
// ===== library types =====

// folder: Library/Modbus/Core/Query

TYPE "mb_set_udt"
   STRUCT
      signed : Bool;   // Set true if it's a signed number.
      double : Bool;   // Get two trailing words (4 bytes) from buffer. False, get one word (2 bytes).
      factor : Real := 1.0;   // Factor the value from the buffer is multiplied with.
   END_STRUCT;
END_TYPE

// folder: Library/Modbus/Core/Sb

TYPE "mb_station_block_udt"
   STRUCT
      conf : Struct   // Configuration
         unit : USInt;   // mb_addr
         skip_code : Bool;   // Skip all code in header and footer fc's.
         disable : Bool;   // Skip all queries
         read_only : Bool;   // Skip all write queries. (fc 5,6,15,16)
         max_comm_error : USInt := 2;   // Repeating erros before communication_error flag is set
         exec_quantity : USInt := 1;   // Number of queries to be exec. at each loop.
      END_STRUCT;
      out : Struct   // Outputs
         Error : Bool;   // All errors, including communication errors
         Communication_error : Bool;   // only communication errors
         Finnish : Bool;   // qid is handed over to next device.
      END_STRUCT;
      log : Struct   // Logging for development and debugging.
         Connected_time : DTL;   // The time the device was connected to the bus
         Disconnected_time : DTL;   // The time, if a device was disconnected to the bus
         Done_cnt : UDInt;   // Successfully queries counter for this device
         Error_comm_cnt : UDInt;   // Communication erros cnt.
         Error_exception_cnt : UDInt;   // Failed queries counter for this device
         Error_status : Word;   // Status code from mb_master or mb_client
         Error_data_addr : UDInt;   // d_addr for last failed querie; handy for troubleshooting
      END_STRUCT;
      z : Struct   // Internal states.
         header_qid : UInt;   // qid value at device header
         comm_err_cnt : USInt;   // Repeating communication errors
         exec_cnt : USInt;   // Numb. of exec. q. this loop
         offset_qid : UInt := 1;   // Device query id.
         err_hold : Bool;   // Help var for .out.error
      END_STRUCT;
   END_STRUCT;
END_TYPE

// folder: Library/Modbus/Core/Tcp

TYPE "mb_tcp_connection_udt"
   STRUCT
      ip : Array[1..4] of USInt;   // IP address
      tcp_port : UInt := 502;
      timeout : Time;
      Error : Bool;
      Error_network : Bool;   // Error with network connection
      Error_unit : USInt;   // Device with error
      z : Struct   // Internal variables
         qid_bellow : Bool;
         disconnect : Bool;   // This tcp-connection has disconnected the connection.
         init_at_header : Bool;   // True if run-state is INIT_QUERY at the header.
      END_STRUCT;
   END_STRUCT;
END_TYPE

// folder: Library/Modbus/Station blocks/sb Untested/M/Mettler

TYPE "mettlerToledoInd560Udt"
   STRUCT
      readMsgSlot : Array[1..4] of Struct
         cmdRespons : Struct
            FP_1 : Bool;
            FP_2 : Bool;
            FP_3 : Bool;
            FP_4 : Bool;
            FP_5 : Bool;
            data_integrity : Bool;
            cmdAck1 : Bool;
            cmdAck2 : Bool;
         END_STRUCT;
         reserved : Byte;   // volt
         data : Real;
         scale_status : Struct
            x08_Enter_Key : Bool;
            x09_Input_1 : Bool;
            x10_Input_2 : Bool;
            x11_Input_3 : Bool;
            x12_Motion : Bool;
            x13_Net_Mode : Bool;
            x14_Data_Integrity_2 : Bool;
            x15_Data_OK : Bool;
            x00_Target_1 : Bool;
            x01_Comparator_1 : Bool;
            x02_Targe_2 : Bool;
            x03_Comparator_2 : Bool;
            x04_Target_3 : Bool;
            x05_Alway_true : Bool;
            x06_TE_bit_1 : Bool;
            x07_TE_bit_2 : Bool;
         END_STRUCT;
      END_STRUCT;
      writeMsgSlot : Array[1..4] of Struct
         cmd : UInt;
         data : Real;
      END_STRUCT;
      run : Struct   // Data calculated from readMsgSlot
         PF : Array[1..4] of USInt;   // Floating point input indication
         cmdAck : Array[1..4] of USInt;
      END_STRUCT;
      occupiedMsgSlots : Array[1..4] of Bool;
      queryDone : Struct
         read : Bool;
         write : Bool;
      END_STRUCT;
   END_STRUCT;
END_TYPE

// folder: Library/Modbus/Station blocks/udt interfaces

TYPE "energy_udt"
   STRUCT
      current : Struct
         L : Array[1..3] of Real;   // A - Live
         N : Real;   // A - Neutral
         avg : Real;   // A - Average
      END_STRUCT;
      voltage : Struct
         L_L : Array[1..3] of Real;   // V
         L_L_avg : Real;   // V - Average
         L_N : Array[1..3] of Real;   // V
         L_N_avg : Real;   // V - Average
      END_STRUCT;
      power : Struct
         active : Struct
            L : Array[1..3] of Real;   // kW
            total : Real;   // kW
         END_STRUCT;
         reactive : Struct
            L : Array[1..3] of Real;   // kVAR
            total : Real;   // kVAR
         END_STRUCT;
         apparent : Struct
            L : Array[1..3] of Real;   // kVA
            total : Real;   // kVA
         END_STRUCT;
      END_STRUCT;
      energy : Struct   // (Accumulated)
         active_out : Real;   // kWh - delivered
         active_in : Real;   // kWh - received
         reactive_out : Real;   // kVARh
         reactive_in : Real;   // kVARh
         apparent_out : Real;   // kVAh
         apparent_in : Real;   // kVAh
      END_STRUCT;
      reverse_phase_order : Bool;
   END_STRUCT;
   // // voltage.L_L[1] : V
END_TYPE

TYPE "variable_frequency_drive_udt"
   STRUCT
      in : Struct   // Input
         ref : Real;   // %
         start : Bool;
         cost : Bool;
         dc_break : Bool;
         quick_stop : Bool;
         reset : Bool;
      END_STRUCT;
      out : Struct   // Output
         ready : Bool;   // Whating only for start signal from plc
         auto : Bool;   // Auto on keypad of device.
         in_operation : Bool;   // Device is operation.
         running : Bool;   // Motor is spinning
         error : Bool;
         power : Real;   // [kW]
         current : Real;   // [A]
         voltage : Real;   // [V]
         frequency : Real;   // [Hz]
         rpm : Real;   // Revolutions per minute
         output_percent : Real;
         torque_percent : Real;
         heatsing_temperature : Real;   // degrees celsius
      END_STRUCT;
   END_STRUCT;
END_TYPE

TYPE "flow_udt"
   STRUCT
      volume_flow : Real;   // kg/s
      mass_flow : Real;   // m3/s
      velocity : Real;   // m/s
      density : Real;   // kg/m3
      temperature : Real;   // °C
   END_STRUCT;
END_TYPE

// folder: Library/Modbus/.Start examples

FUNCTION "mb_Readme" : Void   // FC13, SCL
{ S7_Optimized_Access := 'TRUE' }
VERSION : 0.1
BEGIN
   (* Instructions:

   - Add one of the exmple FB's to your PLC.
   - Call that FB from a cyclic OB.
   - Terminate connection to type on the example FB. (Right click the FB)
   - Set hardware_id, buad-rate, ip, tcp-port, etc, to the correct value.
   - Look inside the library and check if there is a ready station block (SB),
     for your program. If there isn't then a new has to be made. 
   - Station blocks can be single-DB's or multi-instances in a FB.
   - Remove the exmple code and example SB's.

     IMPORTANT: As stated above, the start examples fb, need to be terminated 
     from the library type. If the type is edited and later there is a library 
     update, then all the changes will get lost.

   - Instructions need to be set to the latest version: (Usually already okay)
      * Instructions -> Communication -> Others -> Modbus TCP
      * Instructions -> Communication -> Communication processor -> Modbus
      * Instructions -> Communication -> Communication processor -> Modbus (RTU)  
      * Instructions -> Basic instructions -> Word logic operations -> SEL.
     Change version in the right column.

   *)
END_FUNCTION

// folder: Library/Modbus/.Start examples/Rtu/1200

FUNCTION_BLOCK "modbus_rtu_1200"   // FB104, SCL
{ S7_Optimized_Access := 'TRUE' }
VERSION : 0.1
   VAR
      mb_query : "mb_query";
      mb_rtu1200_ctrl : "mb_rtu1200_ctrl";
      abb_aquaMaster_device1 : "abb_aquaMaster_3";
      abb_aquaMaster_device2 : "abb_aquaMaster_3";
      abb_aquaMaster_device3 : "abb_aquaMaster_3";
      Auma_valve : "Auma_valve";
      Phoenix_Contact_UPS : "Phoenix_Contact_UPS";
      resault_data : Word;
   END_VAR
BEGIN
   // hardware_id: Can be found inside "Device configuration".
   // baud:        Bits per sec. (Parity is even by default)
   // mb_query:    The FB that connects everything together.
   #mb_rtu1200_ctrl(hardware_id := 0, // REPLACE WITH CORRECT ID.
                    baud := 19200,
                    mb_query := #mb_query);

   // - Timeout is calculated automatically.
   // - Each blocks bellow represent one device on the bus.

   // Three Abb aqua-master's.
   #abb_aquaMaster_device1(mb_addr := 1, mb_query := #mb_query);
   #abb_aquaMaster_device2(mb_addr := 2, mb_query := #mb_query);
   #abb_aquaMaster_device3(mb_addr := 3, mb_query := #mb_query);

   // A valve 
   #Auma_valve(mb_addr := 4, mb_query := #mb_query);

   // A UPS.
   #Phoenix_Contact_UPS(mb_addr := 5, mb_query := #mb_query);

   // A station block can be used both for both modbus rtu and tcp. This
   // is particular useful if a tcp-rtu-gateway is used. The same program
   // could be used, just swap mb_master_1200_ctrl, with mb_client_ctrl.

   // Read holding register 456 from device with modbus address 123.
   // This is an example showing that a query does not necessarily need
   // to be part of a station block (SB) as obove, however making
   // reusable SB's is good practice.
   #mb_query(mb_addr := 123,
             mode := #mb_query.c.read.holding_reg,
             data_addr := 456,
             data_ptr := #resault_data);


   // Debugging tip, (no code)
   "mb_Debugging"();
END_FUNCTION_BLOCK

FUNCTION_BLOCK "modbus_rtu_1200_ladder"   // FB114, LAD
TITLE = Example modbus rtu
{ S7_Optimized_Access := 'TRUE' }
VERSION : 0.1
   VAR
      mb_master_ctrl : "mb_rtu1200_ctrl";
      mb_query : "mb_query";
      aquaMaster_device1 : "abb_aquaMaster_3";
      aquaMaster_device2 : "abb_aquaMaster_3";
      Auma_valve : "Auma_valve";
      Phoenix_Contact_UPS : "Phoenix_Contact_UPS";
   END_VAR
   VAR_TEMP   // added for the SCL form of the ladder/FBD networks
      _w1 : Bool;
   END_VAR
BEGIN

REGION Network 1: Modbus master
   // Replace 'hardware_id' with correct id.
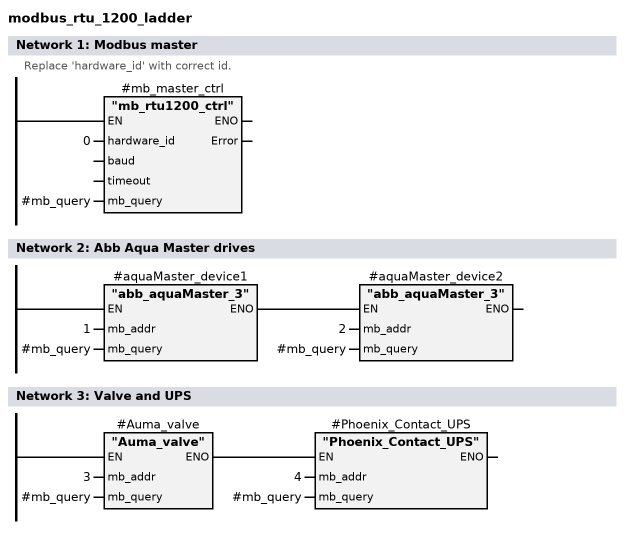
   RUNG wire#powerrail
      #mb_master_ctrl(hardware_id := 0, baud :=, mb_query := #mb_query, Error =>, timeout :=)
   END_RUNG
   // the same network as SCL:
   #mb_master_ctrl(hardware_id := 0, mb_query := #mb_query);   // "mb_rtu1200_ctrl"
END_REGION

REGION Network 2: Abb Aqua Master drives
   RUNG wire#powerrail
      #aquaMaster_device1(mb_addr := 1, mb_query := #mb_query)
      #aquaMaster_device2(mb_addr := 2, mb_query := #mb_query)
   END_RUNG
   // the same network as SCL:
   #aquaMaster_device1(mb_addr := 1, mb_query := #mb_query, ENO => #_w1);   // "abb_aquaMaster_3"
   IF #_w1 THEN
       #aquaMaster_device2(mb_addr := 2, mb_query := #mb_query);   // "abb_aquaMaster_3"
   END_IF;
END_REGION

REGION Network 3: Valve and UPS
   RUNG wire#powerrail
      #Auma_valve(mb_addr := 3, mb_query := #mb_query)
      #Phoenix_Contact_UPS(mb_addr := 4, mb_query := #mb_query)
   END_RUNG
   // the same network as SCL:
   #Auma_valve(mb_addr := 3, mb_query := #mb_query, ENO => #_w1);   // "Auma_valve"
   IF #_w1 THEN
       #Phoenix_Contact_UPS(mb_addr := 4, mb_query := #mb_query);   // "Phoenix_Contact_UPS"
   END_IF;
END_REGION
END_FUNCTION_BLOCK

FUNCTION_BLOCK "modbus_rtu_1200_empty"   // FB119, SCL
{ S7_Optimized_Access := 'TRUE' }
VERSION : 0.1
   VAR
      mb_query : "mb_query";
      mb_master_1200_ctrl : "mb_rtu1200_ctrl";
      _ : Bool;
   END_VAR
BEGIN
   // hardware_id: Can be found inside "Device configuration".
   // baud:        Bits per sec. (Parity is even by default)
   // mb_query:    The FB that connects everything together.
   #mb_master_1200_ctrl(hardware_id := 0, // REPLACE WITH CORRECT ID. ("Local~CB_1241_(RS485)")
                        baud := 19200,
                        mb_query := #mb_query);

   // Timeout is calculated automatically.

   // ... Insert station blocks here ...



   // Debugging tip, (no code)
   "mb_Debugging"();
END_FUNCTION_BLOCK

// folder: Library/Modbus/.Start examples/Rtu/1500

FUNCTION_BLOCK "modbus_rtu_1500_empty"   // FB5, SCL
{ S7_Optimized_Access := 'TRUE' }
VERSION : 0.1
   VAR
      mb_query : "mb_query";
      mb_rtu1500_ctrl : "mb_rtu1500_ctrl";
      _ : Bool;
   END_VAR
BEGIN
   // hardware_id:     May be found inside the hardware configuration.
   // operating_mode:  0: RS232, 2: RS422, 4: RS485.
   // baud:            Bits per sec. (Parity is even by default)
   // mb_query:        The FB that connects everything together.
   #mb_rtu1500_ctrl(hardware_id := 0, // REPLACE WITH CORRECT ID.
                    operating_mode := 4, // RS-485
                    baud := 19200, // bps
                    mb_query := #mb_query);

   // Timeout is calculated automatically.


   // ... Insert station blocks here ...



   // Debugging tip, (no code)
   "mb_Debugging"();
END_FUNCTION_BLOCK

FUNCTION_BLOCK "modbus_rtu_1500_ladder"   // FB97, LAD
TITLE = Example modbus rtu for S7-1500
{ S7_Optimized_Access := 'TRUE' }
VERSION : 0.1
   VAR
      mb_rtu1500_ctrl : "mb_rtu1500_ctrl";
      mb_query : "mb_query";
      aquaMaster_device1 : "abb_aquaMaster_3";
      aquaMaster_device2 : "abb_aquaMaster_3";
      Auma_valve : "Auma_valve";
      Phoenix_Contact_UPS : "Phoenix_Contact_UPS";
   END_VAR
   VAR_TEMP   // added for the SCL form of the ladder/FBD networks
      _w1 : Bool;
   END_VAR
BEGIN

REGION Network 1: Modbus master
   // hardware_id:            Can be found inside "Device configuration". 
   // operating_mode:    0: RS232, 2: RS422, 4: RS485.
   // baud:                         Bits per sec. (Parity is even by default)
   // mb_query:                The FB that connects everything together.
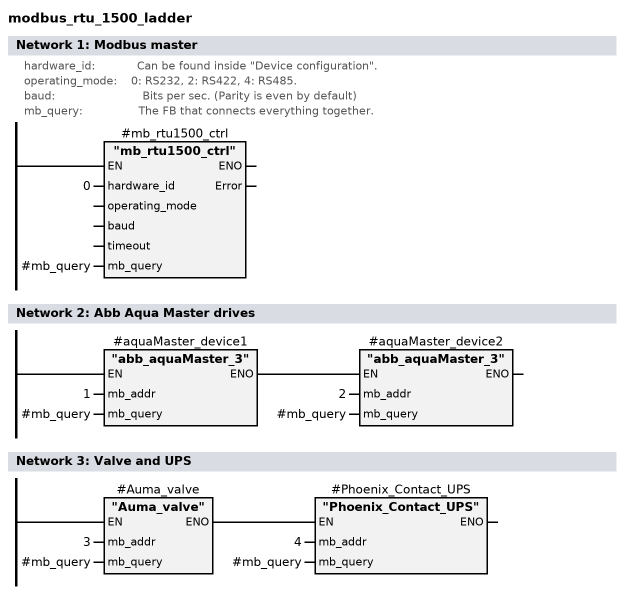
   RUNG wire#powerrail
      #mb_rtu1500_ctrl(hardware_id := 0, operating_mode :=, baud :=, timeout :=, mb_query := #mb_query, Error =>)
   END_RUNG
   // the same network as SCL:
   #mb_rtu1500_ctrl(hardware_id := 0, mb_query := #mb_query);   // "mb_rtu1500_ctrl"
END_REGION

REGION Network 2: Abb Aqua Master drives
   RUNG wire#powerrail
      #aquaMaster_device1(mb_addr := 1, mb_query := #mb_query)
      #aquaMaster_device2(mb_addr := 2, mb_query := #mb_query)
   END_RUNG
   // the same network as SCL:
   #aquaMaster_device1(mb_addr := 1, mb_query := #mb_query, ENO => #_w1);   // "abb_aquaMaster_3"
   IF #_w1 THEN
       #aquaMaster_device2(mb_addr := 2, mb_query := #mb_query);   // "abb_aquaMaster_3"
   END_IF;
END_REGION

REGION Network 3: Valve and UPS
   RUNG wire#powerrail
      #Auma_valve(mb_addr := 3, mb_query := #mb_query)
      #Phoenix_Contact_UPS(mb_addr := 4, mb_query := #mb_query)
   END_RUNG
   // the same network as SCL:
   #Auma_valve(mb_addr := 3, mb_query := #mb_query, ENO => #_w1);   // "Auma_valve"
   IF #_w1 THEN
       #Phoenix_Contact_UPS(mb_addr := 4, mb_query := #mb_query);   // "Phoenix_Contact_UPS"
   END_IF;
END_REGION
END_FUNCTION_BLOCK

FUNCTION_BLOCK "modbus_rtu_1500"   // FB108, SCL
{ S7_Optimized_Access := 'TRUE' }
VERSION : 0.1
   VAR
      mb_query : "mb_query";
      mb_rtu1500_ctrl : "mb_rtu1500_ctrl";
      abb_aquaMaster_device1 : "abb_aquaMaster_3";
      abb_aquaMaster_device2 : "abb_aquaMaster_3";
      abb_aquaMaster_device3 : "abb_aquaMaster_3";
   END_VAR
BEGIN
   // hardware_id:     May be found inside the hardware configuration.
   // operating_mode:  0: RS232, 2: RS422, 4: RS485.
   // baud:            Bits per sec. (Parity is even by default)
   // mb_query:        The FB that connects everything together.
   #mb_rtu1500_ctrl(hardware_id := 0, // REPLACE WITH CORRECT ID.
                    operating_mode := 4, // RS-485
                    baud := 19200, // bps
                    mb_query := #mb_query);

   // Timeout is calculated automatically

   // Each blocks bellow represent one device on the bus. 
   #abb_aquaMaster_device1(mb_addr := 1, mb_query := #mb_query);
   #abb_aquaMaster_device2(mb_addr := 2, mb_query := #mb_query);
   #abb_aquaMaster_device3(mb_addr := 3, mb_query := #mb_query);


   // Debugging tip, (no code)
   "mb_Debugging"();
END_FUNCTION_BLOCK

// folder: Library/Modbus/.Start examples/Tcp

FUNCTION_BLOCK "modbus_tcp_empty"   // FB79, SCL
{ S7_Optimized_Access := 'TRUE' }
VERSION : 0.1
   VAR
      mb_query : "mb_query";
      mb_client_ctrl : "mb_tcp_ctrl";
      ip : Array[1..4] of USInt;
      mb_delay_between_queries : "mb_delay_between_queries";
   END_VAR
BEGIN
   // IP-address of the modbus server
   #ip[1] := 192;
   #ip[2] := 168;
   #ip[3] := 1;
   #ip[4] := 2;

   // interface:  Profinet interface.
   //             (Find const. inside "Device configuration")
   // conn_id:    A unique id for each tcp connectin in the plc.
   // ip_addr:    The ip-address of the server. (Array of 4 bytes)
   // tcp_port:   Default port is 502. (UDP isn't available)
   // timeout:    Depends on the network conncetion.
   // mb_query:   The query FB.
   #mb_client_ctrl(interface := 0, // REPLACE WITH CORRECT ID OR CONST,
                                   // Eg. "Local~PROFINET_interface_1",
                   conn_id := 123,
                   ip_addr := #ip,
                   tcp_port := 502,
                   timeout := T#2s,
                   mb_query := #mb_query);

   // Delay the query execution, this prevent the plc from
   // jamming the network. Adjust the time to the application.
   #mb_delay_between_queries(delay := T#500ms,
                             mb_query := #mb_query);




   // ... Insert station blocks here ...




   // Debugging tip, (no code)
   "mb_Debugging"();
END_FUNCTION_BLOCK

FUNCTION_BLOCK "modbus_tcp_ladder"   // FB98, LAD
TITLE = Example modbus tcp
{ S7_Optimized_Access := 'TRUE' }
VERSION : 0.1
   VAR
      mb_client_ctrl : "mb_tcp_ctrl";
      mb_query : "mb_query";
      mb_delay_between_queries : "mb_delay_between_queries";
      ip : Array[1..4] of USInt;
      siemens_PAC3200 : "Siemens_PAC3200";
   END_VAR
   VAR_TEMP   // added for the SCL form of the ladder/FBD networks
      _w1 : Bool;
   END_VAR
BEGIN

REGION Network 1 (SCL): IP-address
   #ip[1] := 192;
   #ip[2] := 168;
   #ip[3] := 1;
   #ip[4] := 123;
END_REGION

REGION Network 2: Modbus client ctrl
   // - Insert interface constant, eg "Local~PROFINET_interface_1". 
   // - conn_id need to be unique for all tcp connection in the plc.
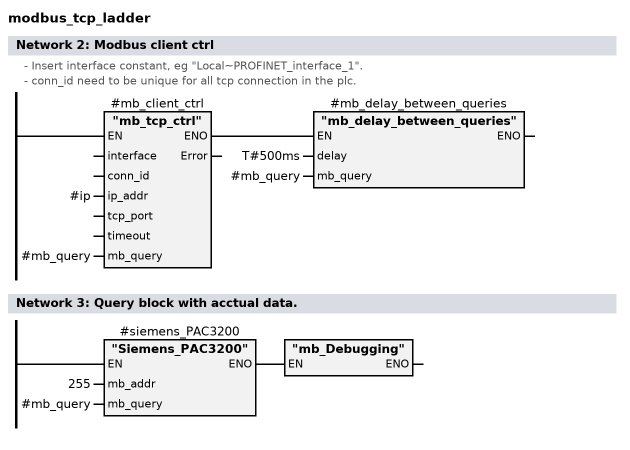
   RUNG wire#powerrail
      #mb_client_ctrl(interface :=, conn_id :=, ip_addr := #ip, tcp_port :=, timeout :=, mb_query := #mb_query, Error =>)
      #mb_delay_between_queries(delay := T#500ms, mb_query := #mb_query)
   END_RUNG
   // the same network as SCL:
   #mb_client_ctrl(ip_addr := #ip, mb_query := #mb_query, ENO => #_w1);   // "mb_tcp_ctrl"
   IF #_w1 THEN
       #mb_delay_between_queries(delay := T#500ms, mb_query := #mb_query);   // "mb_delay_between_queries"
   END_IF;
END_REGION

REGION Network 3: Query block with acctual data.
   RUNG wire#powerrail
      #siemens_PAC3200(mb_addr := 255, mb_query := #mb_query)
      "mb_Debugging"()
   END_RUNG
   // the same network as SCL:
   #siemens_PAC3200(mb_addr := 255, mb_query := #mb_query, ENO => #_w1);   // "Siemens_PAC3200"
   IF #_w1 THEN "mb_Debugging"(); END_IF;
END_REGION
END_FUNCTION_BLOCK

FUNCTION_BLOCK "modbus_tcp"   // FB110, SCL
{ S7_Optimized_Access := 'TRUE' }
VERSION : 0.1
   VAR
      mb_query : "mb_query";
      mb_tcp_ctrl : "mb_tcp_ctrl";
      siemens_PAC3200 : "Siemens_PAC3200";
      ip : Array[1..4] of USInt;
      mb_delay_between_queries : "mb_delay_between_queries";
   END_VAR
BEGIN
   // IP-address of the modbus server
   #ip[1] := 192;
   #ip[2] := 168;
   #ip[3] := 1;
   #ip[4] := 2;

   // interface:  Profinet interface.
   //             (Find const. inside "Device configuration")
   // conn_id:    A unique id for each tcp connectin in the plc.
   // ip_addr:    The ip-address of the server. (Array of 4 bytes)
   // tcp_port:   Default port is 502. (UDP isn't available)
   // timeout:    Depends on the network conncetion.
   // mb_query:   The query FB.
   #mb_tcp_ctrl(interface := 0, // REPLACE WITH CORRECT ID OR CONST,
                // Eg. "Local~PROFINET_interface_1",
                conn_id := 123,
                ip_addr := #ip,
                tcp_port := 502,
                timeout := T#2s,
                mb_query := #mb_query);

   // Delay the query execution, this prevent the plc from
   // jamming the network. Adjust the time to the application.
   #mb_delay_between_queries(delay := T#500ms, mb_query := #mb_query);

   #siemens_PAC3200(mb_query := #mb_query);


   // Debugging tip, (no code)
   "mb_Debugging"();
END_FUNCTION_BLOCK

// folder: Library/Modbus/.Start examples/Tcp/multi_client

FUNCTION_BLOCK "multi_client"   // FB111, SCL
{ S7_Optimized_Access := 'TRUE' }
VERSION : 0.1
   VAR
      ctrl : "mb_tcp_ctrl";
      query : "mb_query";
      delay_between_queries : "mb_delay_between_queries";
      c1 : "mb_tcp_connection_udt";
      c2 : "mb_tcp_connection_udt";
      c3 : "mb_tcp_connection_udt";
      c4 : "mb_tcp_connection_udt";
      c5 : "mb_tcp_connection_udt";
      power_meter_1 : "Siemens_PAC3200";
      power_meter_2 : "Siemens_PAC3200";
      flow_meter_1 : "Siemens_MAG_6000";
      flow_meter_2 : "Siemens_MAG_6000";
      Level_1 : "Mjk_expert";
      Level_2 : "Mjk_expert";
      Level_3 : "Mjk_expert";
   END_VAR
BEGIN
   // This feature is foremost intended for S7-1200 where the number of tcp
   // connections is limited. Another use case it's to get data from hundreds or 
   // even tunsens of devices, and it's then also applicable for S7-1500 plc's.
   // One mb_client use much memory, so you would save memory by using this
   // approach, compare using a client for each connection.
   //
   // One mb_client is connecting and disconnecting to different ip-addresses,
   // and therefore only occupy one connection. The downside with this solution
   // is the delays for data to come in. The library is smart, and it wouldn't
   // waste time on polling devices that has got timeout before.

   // Important: Don't assign anything to #ctrl.ip_addr and #ctrl.tcp_port, when
   //            the library is used in this mode.

   // interface:  Profinet interface. (Find const. inside "Device configuration")
   // conn_id:    A unique id for each tcp connectin in the plc.
   // timeout:    Establish a tcp-connection may take quite long, several
   //             seconds for some devices, so make sure to not set it to short.
   // mb_query:   The query FB.
   #ctrl(interface := 64, conn_id := 123, timeout := T#2s, mb_query := #query);

   // Delay the query execution, this prevent the plc from
   // jamming the network. Adjust the time to the application.
   #delay_between_queries(delay := T#20ms, mb_query := #query);

   REGION TCP-connection 1
       #c1.ip[1] := 192;
       #c1.ip[2] := 168;
       #c1.ip[3] := 0;
       #c1.ip[4] := 2;
       "mb_tcp_connection_header"(conn := #c1, ctrl := #ctrl, q := #query);

       // Note: For some tcp-devices mb_addr need to be set to 255.
       #power_meter_1(mb_query := #query);

       "mb_tcp_connection_foother"(conn := #c1, ctrl := #ctrl, q := #query);
   END_REGION

   REGION TCP-connection 2
       #c2.ip[1] := 192;
       #c2.ip[2] := 168;
       #c2.ip[3] := 0;
       #c2.ip[4] := 3;
       "mb_tcp_connection_header"(conn := #c2, ctrl := #ctrl, q := #query);

       #power_meter_2(mb_query := #query);

       "mb_tcp_connection_foother"(conn := #c2, ctrl := #ctrl, q := #query);
   END_REGION

   REGION TCP-connection 3
       #c3.ip[1] := 192;
       #c3.ip[2] := 168;
       #c3.ip[3] := 0;
       #c3.ip[4] := 4;
       "mb_tcp_connection_header"(conn := #c3, ctrl := #ctrl, q := #query);

       #flow_meter_1(mb_query := #query);

       "mb_tcp_connection_foother"(conn := #c3, ctrl := #ctrl, q := #query);
   END_REGION

   REGION TCP-connection 4
       #c4.ip[1] := 192;
       #c4.ip[2] := 168;
       #c4.ip[3] := 0;
       #c4.ip[4] := 5;
       "mb_tcp_connection_header"(conn := #c4, ctrl := #ctrl, q := #query);

       #flow_meter_2(mb_query := #query);

       "mb_tcp_connection_foother"(conn := #c4, ctrl := #ctrl, q := #query);
   END_REGION

   REGION TCP-connection 5 (gateway)
       #c5.ip[1] := 192;
       #c5.ip[2] := 168;
       #c5.ip[3] := 0;
       #c5.ip[4] := 6;
       "mb_tcp_connection_header"(conn := #c5, ctrl := #ctrl, q := #query);

       // For a gateway, any number of station blocks may be placed between
       // header above and the foother bellow.
       #Level_1(mb_addr := 1, mb_query := #query);
       #Level_2(mb_addr := 2, mb_query := #query);
       #Level_3(mb_addr := 3, mb_query := #query);

       "mb_tcp_connection_foother"(conn := #c5, ctrl := #ctrl, q := #query);
   END_REGION

   "mb_Debugging"(); // Just text.
END_FUNCTION_BLOCK

FUNCTION_BLOCK "multi_client_empty"   // FB118, SCL
{ S7_Optimized_Access := 'TRUE' }
VERSION : 0.1
   VAR
      ctrl : "mb_tcp_ctrl";
      query : "mb_query";
      delay_between_queries : "mb_delay_between_queries";
      c1 : "mb_tcp_connection_udt";
      c2 : "mb_tcp_connection_udt";
      c3 : "mb_tcp_connection_udt";
   END_VAR
BEGIN

   // interface:  Profinet interface. (Find const. inside "Device configuration")
   // conn_id:    A unique id for each tcp connectin in the plc.
   // timeout:    Establish a tcp-connection may take quite long, serveral
   //             secounds for some devices, so make sure to not set it to short.
   //             On the other hand it's also important to set it too long.
   //             On a local network you may try to start with 3 sec.
   // mb_query:   The query FB.                                     
   #ctrl(interface := 64, conn_id := 123, timeout := T#3s, mb_query := #query);

   // Delay the query execution, this prevent the plc from
   // jamming the network. Adjust the time to the application.
   #delay_between_queries(delay := T#50ms, mb_query := #query);

   REGION TCP-connection 1
       #c1.ip[1] := 192;
       #c1.ip[2] := 168;
       #c1.ip[3] := 0;
       #c1.ip[4] := 0;
       "mb_tcp_connection_header"(conn := #c1, ctrl := #ctrl, q := #query);

       // Insert sb here.

       "mb_tcp_connection_foother"(conn := #c1, ctrl := #ctrl, q := #query);
   END_REGION

   REGION TCP-connection 2
       #c2.ip[1] := 192;
       #c2.ip[2] := 168;
       #c2.ip[3] := 0;
       #c2.ip[4] := 0;
       "mb_tcp_connection_header"(conn := #c2, ctrl := #ctrl, q := #query);

       // Insert sb here.

       "mb_tcp_connection_foother"(conn := #c2, ctrl := #ctrl, q := #query);
   END_REGION

   REGION TCP-connection 3
       #c3.ip[1] := 192;
       #c3.ip[2] := 168;
       #c3.ip[3] := 0;
       #c3.ip[4] := 0;
       "mb_tcp_connection_header"(conn := #c3, ctrl := #ctrl, q := #query);

       // Insert sb here.

       "mb_tcp_connection_foother"(conn := #c3, ctrl := #ctrl, q := #query);
   END_REGION


   "mb_Debugging"(); // Only text
END_FUNCTION_BLOCK

FUNCTION_BLOCK "multi_client_array"   // FB121, SCL
{ S7_Optimized_Access := 'TRUE' }
VERSION : 0.1
   VAR
      ctrl : "mb_tcp_ctrl";
      query : "mb_query";
      delay_between_queries : "mb_delay_between_queries";
      c : Array[2..50] of "mb_tcp_connection_udt";
      power_meter : Array[2..50] of "Siemens_PAC3200";
      j : Int := 2;
   END_VAR
BEGIN
   // An example with many tcp devices.

   // interface:  Profinet interface. (Find const. inside "Device configuration")
   // conn_id:    A unique id for each tcp connectin in the plc.
   // timeout:    Establish a tcp-connection may take quite long, serveral
   //             secounds for some devices, so make sure to not set it to short. 
   // mb_query:   The query FB.                                     
   #ctrl(interface := 64, conn_id := 123, timeout := T#2s, mb_query := #query);

   // Delay the query execution, this prevent the plc from
   // jamming the network. Adjust the time to the application.
   #delay_between_queries(delay := T#20ms, mb_query := #query);

   #c[#j].ip[1] := 192;
   #c[#j].ip[2] := 168;
   #c[#j].ip[3] := 0;
   #c[#j].ip[4] := INT_TO_USINT(#j);
   "mb_tcp_connection_header"(conn := #c[#j], ctrl := #ctrl, q := #query);

   #power_meter[#j]power_meter(mb_query := #query);

   "mb_tcp_connection_foother"(conn := #c[#j], ctrl := #ctrl, q := #query);

   #j += BOOL_TO_INT(#power_meter[#j].sb.out.Finnish);
   IF #j > 50 THEN
       #j := 2;
   END_IF;

   "mb_Debugging"(); // Just text.
END_FUNCTION_BLOCK

// folder: Library/Modbus/Core/Ctrl

FUNCTION_BLOCK "mb_tcp_ctrl"   // FB9, SCL
{ S7_Optimized_Access := 'TRUE' }
VERSION : 1.0
   VAR_INPUT
      interface : Hw_Any := 64;   // Profinet interface id
      conn_id : Conn_Ouc := 123;   // Connection id. Should be unique between all tcp connections.
      ip_addr : Array[1..4] of USInt;   // IPv4 address.
      tcp_port : UInt := 502;
      timeout : Time := T#3s;
   END_VAR
   VAR_OUTPUT
      Error : Bool;   // error flag with tof timer
   END_VAR
   VAR_IN_OUT
      mb_query : "mb_query";   // udt mb
   END_VAR
   VAR
      conf : Struct   // Configuration that normal shouldn't need to be changed.
         disconnect : Bool := false;
         retries : USInt := 0;
         timeout_connect : Time;   // May be set longer, then the main timeout. T#0s => Use normal timeout.
         disconnect_on_80A3 : Bool := true;
         fast_err : Bool := true;
      END_STRUCT;
      client : MB_CLIENT;
      tcon_ip_v4 : TCON_IP_v4;
      tdiscon : TDISCON;
      ton_timeout : TON_TIME;
      end : "mb_internal_e";
      override_timeout : Time;
      connected_memory : Bool;
      connected : Bool;
   END_VAR
   VAR_TEMP
      comm_err : Bool;
      c : SInt;
      t : Time;   // Timeout
   END_VAR
   VAR CONSTANT
      INIT_QUERY : USInt := 2;
      EXEC_QUERY : USInt := 3;
   END_VAR
BEGIN
   // Rexhip - Extended modbus library.
   //
   // Modbus tcp for S7-1200 and S7-1500.

   REGION Init
       // InterfaceId can be found inside "Device configuration".
       #tcon_ip_v4.InterfaceId := #interface;
       #tcon_ip_v4.ID := #conn_id; // Connection id
       FOR #c := 1 TO 4 DO // usint easier to read ip in plc-monitoring.
           #tcon_ip_v4.RemoteAddress.ADDR[#c] := USINT_TO_BYTE(#ip_addr[#c]); 
       END_FOR;
       #tcon_ip_v4.RemotePort := #tcp_port;
       #tcon_ip_v4.ConnectionType := 11; // tcp
       #tcon_ip_v4.ActiveEstablished := true; // Client

       IF #conf.disconnect THEN // Reset memory
           #connected_memory := false;  
       END_IF;

       IF #mb_query.z.run.state = #INIT_QUERY THEN
           RESET_TIMER(#ton_timeout);

           // Conversion of function codes.     
           "mb_internal_a"(Mode => #client.MB_MODE,
                           Data_addr => #client.MB_DATA_ADDR,
                           mb_query := #mb_query);
           #client.MB_Unit_ID := UINT_TO_BYTE(#mb_query.z.q.mb_addr);
           #client.Retries := #conf.retries;
           // Reset all stat-flags.
           #mb_query.stat.error := #mb_query.stat.error_comm :=
           (* *)#mb_query.stat.done := false;

           #mb_query.z.run.state := #EXEC_QUERY; // Next state.
       END_IF;
   END_REGION

   REGION Timeout
       IF #override_timeout <> T#0s THEN
           // If a value has been set for multi connection.
           #t := #override_timeout;
           #override_timeout := T#0s;
       ELSE
           // Use #timeout if #timeout_connect is set to zero. 
           // and connection has not been established before.
           #t := SEL(G := #conf.timeout_connect <> T#0s
                     AND NOT #connected_memory,
                     IN0 := #timeout,
                     IN1 := #conf.timeout_connect);
       END_IF;
       #t := LIMIT(MN := t#100ms, IN := #t, MX := t#10S);
       // If mb_client does not establish a connection it will not throw
       // timeout error. Timeout is handled manually for that case. 
       PRESET_TIMER(PT := #t,
                    TIMER := #ton_timeout);
       #client.Rcv_Timeout := UDINT_TO_REAL(T_CONV(#t)) * 0.001;
       #ton_timeout(IN := #mb_query.z.run.state = #EXEC_QUERY,
                    PT := #ton_timeout.PT);
   END_REGION

   REGION Exec            
       // STATUS 16#80A3 : 
       // If a new download has taken place, and this block is re-initialize,
       // then the mb_client block will output the error code saying that:
       // "Attempt being made to re-establish an existing connection." The
       // solution to this problem is to disconnect and then reconnect. It
       // dosen't work to use disconnect input on the mb_client block.
       #tdiscon(REQ := #client.STATUS = 16#80A3 AND #conf.disconnect_on_80A3,
                ID := #conn_id);

       #client(DISCONNECT := #conf.disconnect OR #tdiscon.BUSY,
               REQ := #mb_query.z.run.state = #EXEC_QUERY
               AND NOT #client.BUSY
               AND NOT #client.DISCONNECT
               AND #client.Connected
               AND NOT #ton_timeout.Q,
               MB_MODE := #client.MB_MODE,
               MB_DATA_ADDR := #mb_query.z.q.data_addr,
               MB_DATA_LEN := #mb_query.z.q.data_len,
               BUSY => #mb_query.stat.busy,
               STATUS => #mb_query.stat.status,
               MB_DATA_PTR := #mb_query.z.buffer,
               CONNECT := #tcon_ip_v4);

       IF #mb_query.z.run.state = #EXEC_QUERY
           AND NOT #client.BUSY
           AND #connected = #client.Connected
           // Disconnect hasn't change the last cycle.
           AND #mb_query.stat.status <> 16#80A7
           // 80A7: TDISCON executed before TCON had completed.
           // This error may happen if connection is not achieved,
           // it need to be blocked from sent to the sb's.
       THEN
           IF #client.ERROR OR #client.DONE THEN
               #mb_query.stat.error := #client.ERROR;
               #mb_query.stat.done := #client.DONE;
               // Comm. error and timeout handeling. 
               CASE WORD_TO_UINT(#mb_query.stat.status) OF
                   16#80C8, // No response from the server.
                   16#818C: // blocked_proc_timeout or rcv_timeout.
                       #comm_err := true;
               END_CASE;
               #mb_query.stat.error_comm := #comm_err OR NOT #client.Connected;
           ELSIF #ton_timeout.Q THEN
               #mb_query.stat.error := #mb_query.stat.error_comm := true;
               #mb_query.stat.done := false;
           END_IF;
       END_IF;
       #connected := #client.Connected;
       IF #client.Connected THEN
           #connected_memory := true;
       END_IF;
   END_REGION

   // End is a comman FB for both tcp and rtu.
   #end(mb_query := #mb_query, Error => #Error);

   // Set error flags on all sb's.
   IF NOT #client.Connected
       AND #conf.fast_err
       AND NOT #client.DISCONNECT  // Cmd connect
       AND (#connected_memory OR #ton_timeout.Q) // - Connection established
   THEN                                          //   before or timeout.
       #mb_query.z.sb.set_err := true; 
   END_IF;
END_FUNCTION_BLOCK

FUNCTION_BLOCK "mb_rtu1500_ctrl"   // FB10, SCL
{ S7_Optimized_Access := 'TRUE' }
VERSION : 1.0
   VAR_INPUT
      hardware_id : Port;   // hardware id
      operating_mode : USInt := 4;   // 0: RS232, 2: RS422, 4: RS485.
      baud : UDInt := 19200;   // Bits per sec.
      timeout : Time := T#400ms;   // Automatically calculated if set to zero. (T#0s)
   END_VAR
   VAR_OUTPUT
      Error : Bool;   // One or more errors in the whole application.
   END_VAR
   VAR_IN_OUT
      mb_query : "mb_query";
   END_VAR
   VAR
      conf : Struct   // Configuration that normal shouldn't need to be changed.
         parity : UInt := 2;   // 0=no-parity, 1=odd, 2=even.
         retries : USInt := 0;
      END_STRUCT;
      comm_load : Modbus_Comm_Load;
      leader : Modbus_Master;
      buffer : "mb_internal_b";
      end : "mb_internal_e";
      comm_load_done : Bool;
      init_hw : Bool := true;
   END_VAR
   VAR CONSTANT
      INIT_QUERY : USInt := 2;
      EXEC_QUERY : USInt := 3;
      RECIVE_RESUALT : USInt := 4;
   END_VAR
BEGIN
   // Rexhip - Extended modbus library.
   //
   // RTU leader for S7-1500
   // 
   // This master blocks works for both S7-1200 and S7-1500. For S7-1200
   // it's recommended to use the other ctrl block, mb_master_1200_ctrl
   // because it use less memory. Please read the documentation, before
   // dive into the code bellow.

   REGION Init
       IF #init_hw THEN  // (true on first_scan)
           #comm_load.RESP_TO := T_CONV(#timeout)
           + UDINT_TO_UINT(4500000 / #baud);
       END_IF;
       // Initiate the hardware.
       #comm_load.RETRIES := #conf.retries;
       #comm_load.MODE := #operating_mode;
       #comm_load(REQ := #init_hw,
                  PORT := #hardware_id,
                  BAUD := #baud,
                  PARITY := #conf.parity, // Even is default.
                  RESP_TO := #comm_load.RESP_TO,
                  MB_DB := #leader.MB_DB);
       #init_hw := false; // Hw init Finnised
       IF #comm_load.DONE THEN
           #comm_load_done := true;
       END_IF;

       IF #mb_query.z.run.state = #INIT_QUERY THEN
           // Modicon convention address conversion.
           "mb_internal_a"(Mode => #leader.MODE,
                           Data_addr => #leader.DATA_ADDR,
                           mb_query := #mb_query);
          // Copy buffer to a non optimiced memory area.
           IF #mb_query.z.run.write THEN
               #buffer.buffer := #mb_query.z.buffer;
           END_IF;
           IF #comm_load_done THEN
               #mb_query.z.run.state := #EXEC_QUERY;
           ELSE
               // Skip query exec. if init hw didn't go well.
               // The state RECIVE_RESUALT is inside mb_query.
               #mb_query.z.run.state := #RECIVE_RESUALT;
               #mb_query.stat.done := false;
               #mb_query.stat.error := true;
               #mb_query.stat.error_comm := true;
               #mb_query.stat.status := #comm_load.STATUS;
           END_IF;
       END_IF;
   END_REGION

   REGION Exec
       #leader(REQ := #mb_query.z.run.state = #EXEC_QUERY
            AND NOT #leader.BUSY,
            MB_ADDR := #mb_query.z.q.mb_addr,
            MODE := #leader.MODE,
            DATA_ADDR := #leader.DATA_ADDR,
            DATA_LEN := #mb_query.z.q.data_len,
            BUSY => #mb_query.stat.busy,
            DATA_PTR := #buffer.buffer);

       IF #mb_query.z.run.state = #EXEC_QUERY THEN
           #mb_query.stat.error := #leader.ERROR;
           #mb_query.stat.done := #leader.DONE;
           #mb_query.stat.status := #leader.STATUS;
           "mb_internal_f"(buffer := #buffer, mb_query := #mb_query);
       END_IF;
   END_REGION

   // End is a comman FB for both tcp and rtu.
   #end(mb_query := #mb_query, Error => #Error);
END_FUNCTION_BLOCK

FUNCTION_BLOCK "mb_rtu1200_ctrl"   // FB90, SCL
{ S7_Optimized_Access := 'TRUE' }
VERSION : 1.0
   VAR_INPUT
      hardware_id : Port := 0;   // Hardware id
      baud : UDInt := 19200;   // Bits per second
      timeout : Time := T#200ms;   // Additional time for timeout, added to the calculated value
   END_VAR
   VAR_OUTPUT
      Error : Bool;   // One or more errors in the whole application.
   END_VAR
   VAR_IN_OUT
      mb_query : "mb_query";
   END_VAR
   VAR
      conf : Struct   // Configuration that normal shouldn't need to be changed.
         parity : UInt := 2;   // 0=no-parity, 1=odd, 2=even.
         retries : USInt := 0;
      END_STRUCT;
      comm_load : MB_COMM_LOAD;
      leader : MB_MASTER;
      buffer : "mb_internal_b";
      end : "mb_internal_e";   // FB common for both rtu and tcp.
   END_VAR
   VAR_TEMP
      tmp_err : Bool;
   END_VAR
   VAR CONSTANT
      INIT_QUERY : USInt := 2;
      EXEC_QUERY : USInt := 3;
      RECIVE_RESUALT : USInt := 4;
   END_VAR
BEGIN
   // Rexhip - Extended modbus library.
   // 
   // RTU leader for S7-1200
   // 
   // This FB use less memory then mb_master_1500_ctrl, but it only works for
   // S7-1200 PLC's. Please read the documentation, before dive into the code
   // bellow. See link in mb_query() FB.

   REGION Init
       IF #mb_query.z.run.state = #INIT_QUERY THEN
           // Modicon convention address conversion.
           "mb_internal_a"(Mode => #leader.MODE,
                           Data_addr => #leader.DATA_ADDR,
                           mb_query := #mb_query);
           // Copy buffer to a non optimiced memory area.
           IF #mb_query.z.run.write THEN
               #buffer.buffer := #mb_query.z.buffer;
           END_IF;
           // Automatically adjust timeout.
           #comm_load.RESP_TO := T_CONV
           ("mb_timeout_rtu_calc"(timeout := #timeout,
                                   baud := #baud,
                                   mb_query := #mb_query));
           #comm_load.RETRIES := #conf.retries;
       END_IF;

       // Initiate the hardware
       #comm_load(REQ := #mb_query.z.run.state = #INIT_QUERY,
                  PORT := #hardware_id,
                  BAUD := #baud,
                  PARITY := #conf.parity, // Even is default
                  RESP_TO := #comm_load.RESP_TO,
                  MB_DB := #leader);

       IF #mb_query.z.run.state = #INIT_QUERY THEN
           IF #comm_load.DONE THEN
               #mb_query.z.run.state := #EXEC_QUERY;
           ELSE
               // Skip query exec. if init hw didn't go well.
               // The state RECIVE_RESUALT is inside mb_query.
               #mb_query.z.run.state := #RECIVE_RESUALT;
               #mb_query.stat.done := false;
               #mb_query.stat.error := #mb_query.stat.error_comm := true;
               #mb_query.stat.status := #comm_load.STATUS;
           END_IF;
       END_IF;
   END_REGION

   REGION Exec        
       #leader(REQ := #mb_query.z.run.state = #EXEC_QUERY
               AND NOT #leader.BUSY,
               MB_ADDR := #mb_query.z.q.mb_addr,
               MODE := #leader.MODE,
               DATA_ADDR := #leader.DATA_ADDR,
               DATA_LEN := #mb_query.z.q.data_len,
               BUSY => #mb_query.stat.busy,
               DATA_PTR := #buffer.buffer);

       IF #mb_query.z.run.state = #EXEC_QUERY THEN
           #mb_query.stat.error := #leader.ERROR;
           #mb_query.stat.done := #leader.DONE;
           #mb_query.stat.status := #leader.STATUS;
           "mb_internal_f"(buffer := #buffer, mb_query := #mb_query);
       END_IF;
   END_REGION

   // End is a comman FB for both tcp and rtu.
   #end(mb_query := #mb_query, Error => #Error);
END_FUNCTION_BLOCK

// folder: Library/Modbus/Core/Other

FUNCTION_BLOCK "search_device"   // FB41, SCL
{ S7_Optimized_Access := 'TRUE' }
VERSION : 0.1
   VAR_OUTPUT
      Done : Bool;
      No_finding : Bool;
   END_VAR
   VAR_IN_OUT
      start_search : Bool;
      mb_addr : UInt;
      mb_query : "mb_query";
   END_VAR
   VAR
      reset_at_start : Bool;
      data_addr : UDInt;
      _ : Bool;
      rtirg_start : R_TRIG;
      resualt_data : Word;
   END_VAR
BEGIN
   #rtirg_start(CLK := #start_search);
   IF #rtirg_start.Q AND #reset_at_start THEN
       #mb_addr := 1;
   END_IF;

   IF #start_search THEN
       #Done := false;
       #No_finding := false;
       #mb_query(mb_addr := #mb_addr,
                 mode := #mb_query.c.read.holding_reg,
                 data_addr := #data_addr,
                 data_ptr := #resualt_data);
       IF #mb_query.Done
           OR #mb_query.Error AND NOT #mb_query.stat.error_comm
       THEN
           #Done := true;
           #start_search := false;
       ELSIF #mb_query.Error THEN
           IF #mb_addr < 247 THEN
               #mb_addr += 1;
           ELSE
               #No_finding := true;
               #start_search := false;
           END_IF;
       END_IF;
   END_IF;
END_FUNCTION_BLOCK

FUNCTION_BLOCK "mb_watchdog"   // FB122, SCL
{ S7_Optimized_Access := 'TRUE' }
VERSION : 0.1
   VAR_INPUT
      pt : Time := T#12s;   // Need to be larger then timeout.
   END_VAR
   VAR_OUTPUT
      Error : Bool;
      Status : Word;
      Error_cnt : UDInt;
   END_VAR
   VAR_IN_OUT
      mb_query : "mb_query";
   END_VAR
   VAR
      stat_error : Bool;
      "timer" : TON_TIME;
      old_state : USInt;
      timer_mem : Bool;
      old_q : Bool;
      cnt : UDInt;
   END_VAR
BEGIN
   // Watchdog for modbus library.

   // If state dosen't change for a certain time, then there is
   // a software bug.
   #"timer"(IN := #mb_query.z.run.state = #old_state, PT := #pt);

   IF #"timer".Q AND NOT #timer_mem THEN
       #timer_mem := #stat_error := true;
       #Status := #mb_query.stat.status;
       #Error_cnt := #cnt += 1;
   ELSIF #"timer".Q AND NOT #old_q THEN
       #Error_cnt := #cnt += 1;
   END_IF;

   // Forward the error to the ctrl, so the error flag is set there.
   IF #stat_error THEN
       #mb_query.stat.error := #mb_query.z.sb.error := true;
   END_IF;

   #old_state := #mb_query.z.run.state;
   #old_q := #"timer".Q;
   #Error := #stat_error;
END_FUNCTION_BLOCK

FUNCTION "mb_dataptr_eq_buffer" : Bool   // FC8, SCL
{ S7_Optimized_Access := 'TRUE' }
VERSION : 0.1
   VAR_IN_OUT
      data_ptr : Variant;
      mb_query : "mb_query";
   END_VAR
   VAR_TEMP
      tmp_buffer : Array[0..249] of Byte;
      pos : DInt;
      c : Int;
      "e" : Int;
   END_VAR
BEGIN
   // Most use cases will not need this function !
   // Example:
   // 
   // #mb_query(mb_addr := 123,
   //           mode := #mb_query.c.write.holding_reg,
   //           data_addr := 456,
   //           data_ptr := #data);
   //
   // IF #mb_query.Done AND
   //     "mb_dataPtr_eq_buffer"(data_ptr := #data, mb_query := #mb_query)
   // THEN
   //      // If there are for some reason two write queries that has exatly
   //      // the same parameters, then the Done-flag may not be enough to
   //      // determine which query has been executed. To compare data as
   //      // well, data_ptr to the buffer, then this use this function. It
   //      // will return true if the content is the same.
   // END_IF;
   //
   // ------- 

   #mb_dataptr_eq_buffer := true; // Init. value

   #"e" := Serialize(SRC_VARIABLE := #data_ptr,
                   DEST_ARRAY => #tmp_buffer,
                   POS := #pos);

   // Looking for differences.
   FOR #c := 0 TO #pos - 1 DO
       IF #tmp_buffer[#c] <> #mb_query.z.buffer[#c] THEN
           #mb_dataptr_eq_buffer := false;
           EXIT;
       END_IF;
   END_FOR;
END_FUNCTION

FUNCTION "mb_execute" : Bool   // FC12, SCL
{ S7_Optimized_Access := 'TRUE' }
VERSION : 0.1
   VAR_IN_OUT
      mb_query : "mb_query";
   END_VAR
   VAR_TEMP
      dommy : Bool;
   END_VAR
   VAR CONSTANT
      EXEC_QUERY : USInt := 3;
   END_VAR
BEGIN
   // Most use cases will not need this function !
   // Example:
   // 
   // IF "mb_execute"(#mb_query) THEN
   //     
   //     // Preparing calculations.
   //     
   //     #mb_query(data_addr := 2, data_ptr := #data);
   // END_IF;
   //
   // Usefull if some CPU demanding calculation need to be done
   // before a write query is inserted. Note that a query can later
   // be aborted, thought mb_execute return true.

   #mb_execute := #mb_query.z.run.qid_cnt + 1 = #mb_query.z.run.qid
   (* *)AND #mb_query.z.run.state <> #EXEC_QUERY
   (* *)AND NOT #mb_query.stat.busy;

   IF NOT #mb_execute THEN
       #mb_query(data_ptr := #dommy);
   END_IF;
END_FUNCTION

// folder: Library/Modbus/Core/Query

FUNCTION_BLOCK "mb_query"   // FB1, SCL
{ S7_Optimized_Access := 'TRUE' }
VERSION : 0.1
   VAR_INPUT
      mb_addr : UInt;   // Device addr. (0 to 247)
      mode : USInt;   // Function code: 1,2,3,4,5,6,15,16. (siemens mode shifted to 200 - 202)
      data_addr : UDInt;   // Data addr. (raw telegram value, 0-65535)
      data_len : UInt;   // Data len. 0=>Auto detect
   END_VAR
   VAR_OUTPUT
      Done : Bool;   // Successful query
      Error : Bool;   // Failed query
   END_VAR
   VAR_IN_OUT
      data_ptr : Variant;   // Bytes and bools has to add up to whole word(s)
   END_VAR
   VAR
      c : Struct   // Constants
         read : Struct   // Read: 1, 2, 3, 4
            discrete_output : USInt := 1;   // 1 (coils)
            discrete_input : USInt := 2;   // 2
            holding_reg : USInt := 3;   // 3
            input_reg : USInt := 4;   // 4
         END_STRUCT;
         write : Struct   // Write: 5, 6, 15, 16
            single_discrete_output : USInt := 5;   // 5 (coil) (when len. is eq. to 1)
            single_holding_reg : USInt := 6;   // 6 (when len. is eq. to 1)
            discrete_output : USInt := 15;   // 15 (coils)
            holding_reg : USInt := 16;   // 16
         END_STRUCT;
         mode : Struct   // Modicon convention addressing. (Eg: hold.reg. start at 40001)
            read : USInt := 200;   // Mode 0 (fc: 1, 2, 3, 4)
            write_single : USInt := 201;   // Mode 1 (fc: 5, 6) (when len. is eq. to 1)
            write : USInt := 202;   // Mode 2 (fc: 15, 16)
         END_STRUCT;
         auto_len : USInt := 0;   // Length based on data_ptr (Used for data_len)
      END_STRUCT;
      conf : Struct   // Configuration
         buffer_handler : Bool := TRUE;   // enable buffer handler
         halt : Bool;   // Halt exec. of queries.
      END_STRUCT;
      stat : Struct   // Status of last executed query
         done : Bool;   // Successfull
         error : Bool;   // Error, including timeout error
         busy : Bool;   // mb_master or mb_client is busy.
         error_comm : Bool;   // communication error (timeout or bad crc)
         status : Word;   // status word of mb_master or mb_client
      END_STRUCT;
      z : Struct   // Internal states
         q : Struct   // Query params
            mb_addr : UInt := 1;   // Station address
            mode : USInt := 0;   // Function code
            data_addr : UDInt;   // Data address
            data_len : UInt := 0;   // Data length
         END_STRUCT;
         run : Struct   // Constantly changing variables
            qid : UInt := 1;   // query id
            qid_cnt : UInt;   // Query id cnt. increase for each query, reset in controller. One loop each scan
            state : USInt;
            bytes : USInt;
            write : Bool;   // A write query is inserted
            discrete : Bool;
         END_STRUCT;
         sb : Struct   // Station block functionality
            sid : UInt;   // Device ID
            sid_halt : Bool;
            sid_cnt : UInt;   // Device id cnt
            sid_retry : UInt := 1;   // Retry device id, qComError
            sid_retry_finished : Bool;
            seq_release : Bool;
            head_insert : Bool;   // Inc. at mb_query on insert
            head_recive : Bool;   // Inc. at mb_query on rec.
            reset : Bool;
            log_data_addr : UDInt;   // Tmp.var. for transf. value to mb_device_footer
            exec_all : Bool;
            set_err : Bool;
            error : Bool;
         END_STRUCT;
         buffer : Array[0..249] of Byte;
      END_STRUCT;
   END_VAR
   VAR_TEMP
      tLen : UInt;
      tPos : DInt;
      tDiscrete : Bool;
      "e" : Int;
      tBuffer : Array[0..249] of Byte;
   END_VAR
   VAR CONSTANT
      ORIGIN : USInt := 0;
      INSERT_QUERY : USInt := 1;
      INIT_QUERY : USInt := 2;
      EXEC_QUERY : USInt := 3;
      RECIVE_RESUALT : USInt := 4;
   END_VAR
BEGIN
   // Rexhip - Extended modbus library 
   // --- --- --- ---
   // License:  MIT-license
   // Author:   Ola Bjørnli
   // Web:      www.rexhip.com
   //           github.com/rexhip/rexhip
   // --- --- --- ---
   // 
   // For autmatic calculation of data_len, mb_query can only count
   // whole bytes. After a query where data_len is specified manually,
   // it need to be set back to automatic.
   // -> #mb_query.data_len := #mb_query.c.auto_len;
   //
   // Please read to the documentation and see the examples, before dive
   // into the code bellow.

   REGION Header            
       #Done := #Error := false;

       // qid_cnt is increased for every query (bellow) and reset back
       // to zero in mb_internal_e. Qid (query id) is increased when a
       // query finnish. A query will execute when qit_cnt = qid. Qid
       // is set back to "1" when all queryies has been executed.
       #z.run.qid_cnt += 1;
       IF #z.run.qid_cnt <> #z.run.qid
           OR #z.run.state = #EXEC_QUERY
           OR #stat.busy // mb_master.busy or mb_client.busy
       THEN
           RETURN;
       END_IF;
   END_REGION

   REGION Pre-calc
       // Is this a discrete query ?
       CASE #mode OF
           1, 2, 5, 15: // Function codes
               #tDiscrete := true;
           200..202:
               CASE #data_addr OF
                   1..19999: // 1..9999, 10001..19999:
                       #tDiscrete := true;
               END_CASE;
       END_CASE;

       // data_len=0 => Automatically calculate the length.
       IF #data_len = 0 THEN
           #"e" := Serialize(SRC_VARIABLE := #data_ptr,
                           DEST_ARRAY => #tBuffer,
                           POS := #tPos);
           #tLen := DINT_TO_UINT
           (* *)(SEL(G := #tDiscrete, IN0 := #tPos / 2, IN1 := #tPos * 8));
       ELSE
           #tLen := #data_len;
       END_IF;
   END_REGION

   // Wait inserting next query if halted, else just continue.
   IF #z.run.state = #ORIGIN AND NOT #conf.halt THEN
       #z.run.state := #INSERT_QUERY;
   END_IF;

   CASE #z.run.state OF
       #INSERT_QUERY: // Transfer query params. to internal variables.
           // Figur out if this is a query that will write to the device.
           CASE #mode OF
               5, 6, 15, 16, 201, 202: // Write fc's.
                   #z.run.write := true;
               ELSE // Read
                   #z.run.write := false;
           END_CASE;
           #z.run.discrete := #tDiscrete;
           #z.run.bytes := UINT_TO_USINT
           (SEL(G := #tDiscrete, IN0 := #tLen * 2, IN1 := #tLen / 8));
           // The params is transfered over to the internal mem. They
           // are later transfered to the modbus master block or the
           // client block.
           #z.q.mb_addr := #mb_addr;
           #z.q.mode := #mode;
           #z.q.data_addr := #data_addr;
           #z.q.data_len := #tLen;
           IF #conf.buffer_handler AND #z.run.write THEN
               // Copy the content of #data_ptr to the buffer.
               #tPos := 0; // Start at the beginning of the buffer.
               #"e" := Serialize(SRC_VARIABLE := #data_ptr,
                               DEST_ARRAY => #z.buffer,
                               POS := #tPos);
           END_IF;
           // A msg. to station block foother FC, a new query has
           // been inserted.
           #z.sb.head_insert := true;
           #z.run.state := #INIT_QUERY; // State inside ctrl block.

       #RECIVE_RESUALT: // Query is finnished. (with or without error)  
           // Make sure that the query resault really belong to this
           // query. This may not be the case if another query before
           // is surrounded by a if-statement.
           IF #z.q.mb_addr = #mb_addr
               AND #z.q.mode = #mode
               AND #z.q.data_addr = #data_addr
               AND #z.q.data_len = #tLen
           THEN
               IF #stat.done // Successfull query (no error)
                   AND NOT #z.run.write  // If it's a read query.
                   AND #conf.buffer_handler
               THEN
                   // Copy the content from the buffer to #data_ptr
                   #tPos := 0; // Start at the beginning of the buffer.
                   #"e" := Deserialize(SRC_ARRAY := #z.buffer,
                                     DEST_VARIABLE => #data_ptr,
                                     POS := #tPos);
               END_IF;
               #Done := #stat.done;
               #Error := #stat.error;
               // Temperary store value, so it can be picked up
               // in the sb footer.
               #z.sb.log_data_addr := #data_addr;
               // Msg. to mb_station_footer.
               #z.sb.head_recive := true;
           END_IF;
           #z.run.qid += 1; // Next query
           #z.run.state := #ORIGIN; // (State before insert, see above)
   END_CASE;
END_FUNCTION_BLOCK

FUNCTION "mb_buffer_get" : Real   // FC3, SCL
{ S7_Optimized_Access := 'TRUE' }
VERSION : 0.1
   VAR_INPUT
      addr : DInt;
   END_VAR
   VAR_IN_OUT
      param : "mb_set_udt";
      q : "mb_query";
   END_VAR
   VAR_TEMP
      tmp : DWord;
      offset : DInt;
   END_VAR
BEGIN
   // Get data from buffer and return a real
   // 
   // This function doesn't work for discrete queries.


   // Calculating buffer offset
   #offset := (#addr - UDINT_TO_DINT(#q.z.q.data_addr)) * 2;
   // Check if #addr is inside the quried range.
   IF #offset < 0
       OR #offset / 2 + BOOL_TO_UINT(#param.double) > #q.z.q.data_len
   THEN
       // Error handling.
       #q.stat.status := 16#fffd;
       #q.Error := #q.stat.error := true;
       #q.Done := #q.stat.done := false;
       #q.z.sb.log_data_addr := DINT_TO_UDINT(#addr);
       #mb_buffer_get := DWORD_TO_REAL(16#ffffffff);
   ELSE
       IF #param.double THEN
           #tmp.%B3 := #q.z.buffer[#offset + 0];
           #tmp.%B2 := #q.z.buffer[#offset + 1];
           #tmp.%B1 := #q.z.buffer[#offset + 2];
           #tmp.%B0 := #q.z.buffer[#offset + 3];
       ELSE
           #tmp.%B1 := #q.z.buffer[#offset + 0];
           #tmp.%B0 := #q.z.buffer[#offset + 1];
       END_IF;
       #mb_buffer_get := #param.factor *
       SEL(G := #param.signed,
           IN0 := UDINT_TO_REAL(DWORD_TO_UDINT(#tmp)),
           IN1 := DINT_TO_REAL(DWORD_TO_DINT(#tmp)));
   END_IF;
END_FUNCTION

FUNCTION "mb_query_bits" : Void   // FC9, SCL
{ S7_Optimized_Access := 'TRUE' }
VERSION : 0.1
   VAR_IN_OUT
      data_ptr : Array[*] of Bool;
      mb_query : "mb_query";
   END_VAR
   VAR_TEMP
      discrete : Bool;
      dommy : Bool;
      lower : DInt;
      upper : DInt;
      bits : UInt;
      bytes : UDInt;   // bytes
   END_VAR
   VAR CONSTANT
      INIT_QUERY : USInt := 2;
      EXEC_QUERY : USInt := 3;
      RECIVE_RESUALT : USInt := 4;
   END_VAR
BEGIN
   // This function may be used when the number of bits dosen't
   // add up to whole bytes, for function codes: 1, 2, 5 and 15. 
   // 
   // data_ptr need to be a one dimensional array of bools.
   // --- --- ---

   REGION Header
       IF #mb_query.z.run.qid_cnt + 1 <> #mb_query.z.run.qid
           OR #mb_query.z.run.state = #EXEC_QUERY
           OR #mb_query.stat.busy
       THEN
           // Skip query, qid will not match qid_cnt and
           // my_query will return.
           #mb_query(data_ptr := #dommy);
           RETURN;
       END_IF;
   END_REGION

   REGION Pre-calc
       // Some preparing calculations.
       CASE #mb_query.mode OF // A discrete query ?
           1, 2, 5, 15:
               #discrete := true;
           200..202:
               CASE #mb_query.data_addr OF
                   1..19999: // 1..9999, 10001..19999
                       #discrete := true;
               END_CASE;
       END_CASE;
       #lower := LOWER_BOUND(ARR := #data_ptr, DIM := 1);
       #upper := UPPER_BOUND(ARR := #data_ptr, DIM := 1);
       #bits := DINT_TO_UINT(#upper - #lower + 1); // Elements in array.

       // Auto data len ?
       IF #mb_query.data_len = #mb_query.c.auto_len THEN
           #bytes := (#bits + 7) / 8; // CEIL()
           #mb_query.data_len := SEL(G := #discrete,
                                     IN0 := (#bits + 15) / 16, // CEIL()
                                     IN1 := #bits);
       ELSE
           #bytes := SEL(G := #discrete,
                         IN0 := #mb_query.data_len * 2, // 1 word -> 2 bytes
                         IN1 := (#mb_query.data_len + 7) / 8); // CEIL()
       END_IF;
   END_REGION

   REGION Run
       // Disable buf.h. inside mb_query.
       #mb_query.conf.buffer_handler := false;

       // Run the query.
       #mb_query(data_ptr := #dommy);

       #mb_query.conf.buffer_handler := true; // Enable buf.h. again.
       #mb_query.data_len := #mb_query.c.auto_len; // Back to auto.
   END_REGION

   REGION Insert & recive
       IF #mb_query.z.run.state = #INIT_QUERY  // Insert query.
           AND #mb_query.z.run.write
       THEN
           // Copy the content from data_ptr to the buffer.
           GATHER_BLK(IN := #data_ptr[#lower],
                      COUNT_OUT := #bytes,
                      OUT => #mb_query.z.buffer[0]);

       ELSIF  #mb_query.Done // The query above.
           AND NOT #mb_query.z.run.write  // A read query
       THEN
           // Copy the content from the buffer to data_ptr.
           SCATTER_BLK(IN := #mb_query.z.buffer[0],
                       COUNT_IN := #bytes,
                       OUT => #data_ptr[#lower]);
       END_IF;
   END_REGION
END_FUNCTION

FUNCTION "mb_query_range" : Bool   // FC22, SCL
{ S7_Optimized_Access := 'TRUE' }
VERSION : 0.1
   VAR_INPUT
      start : UInt;   // Start address
      end : DInt;   // End address
   END_VAR
   VAR_IN_OUT
      q : "mb_query";
   END_VAR
   VAR_TEMP
      dommy : Bool;
   END_VAR
   VAR CONSTANT
      EXEC_QUERY : USInt := 3;
   END_VAR
BEGIN
   // Query a range of register

   IF #q.z.run.qid_cnt + 1 = #q.z.run.qid
       AND #q.z.run.state <> #EXEC_QUERY
       AND NOT #q.stat.busy 
   THEN
       // Negative end-value means length.
       #q.data_len := DINT_TO_UINT
       (SEL(G := #end < 0,
             IN0 := DINT_TO_UINT(#end) - #start + 1,
             IN1 := ABS(#end)));

       // Disable buffer handler.
       #q.conf.buffer_handler := false;

       // Run query.
       #q(data_addr := #start,
          data_ptr := #dommy,
          Done => #mb_query_range );

       // Back to default values.
       #q.data_len := #q.c.auto_len;
       #q.conf.buffer_handler := true;
   ELSE
       #q(data_ptr := #dommy);
       #mb_query_range := false;
   END_IF;
END_FUNCTION

FUNCTION "mb_read_buffer" : Int   // FC25, SCL
{ S7_Optimized_Access := 'TRUE' }
VERSION : 0.1
   VAR_INPUT
      addr : UDInt;   // data address
   END_VAR
   VAR_IN_OUT
      ptr : Variant;   // Data ptr
      q : "mb_query";   // mb_query
   END_VAR
   VAR_TEMP
      offset : DInt;
      bytes_queried : UInt;
      deser_err : Int;
   END_VAR
BEGIN
   // Read buffer, extract data from part of the buffer.

   IF #q.Done THEN
       // Where to start extract data in the buffer.
       #offset := UDINT_TO_DINT(#addr - #q.z.q.data_addr) * 2;
       // Copy content from buffer to #ptr
       #deser_err := Deserialize(SRC_ARRAY := #q.z.buffer,
                                 DEST_VARIABLE => #ptr,
                                 POS := #offset);
       IF #deser_err <> 0 THEN // Check for deserialize error
           #q.stat.status := INT_TO_WORD(#deser_err);
           GOTO ERROR_HANDLING;
       ELSE 
           // Outside the new quried data.
           IF #offset > #q.z.run.bytes THEN
               #q.stat.status := 16#ffff;
               GOTO ERROR_HANDLING;
           END_IF;
       END_IF;
   END_IF;
   #mb_read_buffer := 0;
   RETURN;
   ERROR_HANDLING:
   #mb_read_buffer := WORD_TO_INT(#q.stat.status);
   #q.Error := #q.stat.error := true;
   #q.Done := #q.stat.done := false;
   #q.z.sb.log_data_addr := #addr;
END_FUNCTION

// folder: Library/Modbus/Core/Sb

FUNCTION "mb_station_block_header" : Void   // FC10, SCL
{ S7_Optimized_Access := 'TRUE' }
VERSION : 1.0
   VAR_IN_OUT
      sb : "mb_station_block_udt";
      mb_query : "mb_query";
   END_VAR
   VAR CONSTANT
      ORIGIN : USInt := 0;
      EXEC_QUERY : USInt := 3;
   END_VAR
BEGIN
   // Rexhip - Extended modbus library.

   // Please read to the documentation and see the examples, before dive
   // into the code bellow.

   // This block should be called before all queries in a station block.

   // Skip everything !
   IF #sb.conf.skip_code THEN
       RETURN;
   END_IF;

   #mb_query.data_len := 0; // Default is auto-length.
   #mb_query.conf.buffer_handler := true;
   #mb_query.mb_addr := #sb.conf.unit;

   // If device blocks are executeded in diffrent order, a wide wind
   // up effect will occur, (in same OB) this will prevent that.
   IF #mb_query.z.sb.reset THEN
       #sb.z.header_qid := #mb_query.z.run.qid_cnt + 1;
   END_IF;

   // Device id cnt. The first device has id "1". Increased in every
   // mb_device_header, reseted in mb_client_ctrl or mb_master_ctrl.
   #mb_query.z.sb.sid_cnt += 1;

   // mb_query set the same bellow variables to true, at insert or recive.
   // This informastion is later used at the footer.
   #mb_query.z.sb.head_insert := false;
   #mb_query.z.sb.head_recive := false;

   // Reset order, a variable that makes queries in a sb execute in order.
   // #mb_query.z.sb.order := false;

   // When #mb.mb.q.qid = #mb.mb.run.qid_cnt => "This" device has the
   // query-token !
   // - If the query-token points at this device header, or it point to a
   //   query in the previous device, that is surrounded by a if-statement
   //   and the statement is now false.
   // - A gid change can only be done if not "busy", this is to avoid a
   //   resualt from one query being intercepted by another
   IF #mb_query.z.run.qid > #mb_query.z.run.qid_cnt
       AND #mb_query.z.run.qid <= #sb.z.header_qid
       AND #mb_query.z.run.state <> #EXEC_QUERY
       AND NOT #mb_query.stat.busy
   THEN
       // Reset.
       // Go back to the first state in mb_query. New query param. will
       // owerwrite old once.
       #mb_query.z.run.state := #ORIGIN;

       // At first the offset_qid points at the first query of this
       // device. When it has executed the offset will point at the
       // second query. When all queries has executed the offset will
       // be reset back to the first query. (footer) 
       #mb_query.z.run.qid :=
       (* *)#sb.z.header_qid + #sb.z.offset_qid;

       // Order is a variable that makes queries in sb execute in order.
       //    #mb_query.z.sb.order := true;
   END_IF;

   // - The code below is reduce the impact of setting a if-statement
   //   around queries, by setting the qid_cnt to a fixed value at this 
   //   point.
   // - mb_station_block_header will occupy one query-id.  
   #sb.z.header_qid :=
   MAX(IN1 := #mb_query.z.run.qid_cnt + 1,
       IN2 := #sb.z.header_qid);
   #mb_query.z.run.qid_cnt := #sb.z.header_qid;
END_FUNCTION

FUNCTION "mb_station_block_footer" : Void   // FC11, SCL
{ S7_Optimized_Access := 'TRUE' }
VERSION : 1.0
   VAR_IN_OUT
      sb : "mb_station_block_udt";
      mb_query : "mb_query";
   END_VAR
   VAR_TEMP
      "e" : Int;
      err : Bool;
   END_VAR
   VAR CONSTANT
      ORIGIN : USInt := 0;
      INSERT_QUERY : USInt := 1;
   END_VAR
BEGIN
   // Rexhip - Extended modbus library.

   // Please read to the documentation and see the examples, before dive
   // into the code bellow.

   // This fc should be called after all queries in a station block.

   REGION Pre
       IF #sb.conf.skip_code THEN // Skip everything !
           RETURN;
       ELSIF #mb_query.z.sb.set_err THEN
           IF NOT #sb.out.Communication_error THEN
               #"e" := RD_LOC_T(#sb.log.Disconnected_time);
           END_IF;
           #sb.out.Error := #sb.out.Communication_error := #sb.z.err_hold := true;
           #sb.z.comm_err_cnt := 255;
       END_IF;
   END_REGION

   REGION Recive
       IF #mb_query.z.sb.head_recive THEN
           // If there is a query that bellong to this device that has
           // recvied a resault. (with or without error)

           // Counter for exec. queries inside this station block.
           // Default is 1 query for each loop, but may be changed.
           #sb.z.exec_cnt += 1;

           // For application with muliple tcp-settings, is more effectively to
           // execute all queries right away, becouse it's take time to esablish
           // and disconnect tcp connections.
           IF #mb_query.z.sb.exec_all AND #sb.conf.exec_quantity = 1 THEN
               #sb.conf.exec_quantity := 255;
           END_IF;

           // If this is the first succesfylly query after communication error,
           // then log the time this happen. (also exceptions)
           IF #sb.out.Communication_error AND (
               #mb_query.stat.done
               OR #mb_query.stat.error AND NOT #mb_query.stat.error_comm)
           THEN
               #"e" := RD_LOC_T(#sb.log.Connected_time);
           END_IF;

           IF #mb_query.stat.error THEN // Logging - failed query        
               // Store the values for debugging. data_addr will indicate witch 
               // query caused the error, and the status is indicate the error type.
               #sb.log.Error_status := #mb_query.stat.status;
               #sb.log.Error_data_addr := #mb_query.z.sb.log_data_addr;

               // Two counters, one for comm.error and for all other errors.
               IF #mb_query.stat.error_comm THEN
                   #sb.log.Error_comm_cnt += 1; // Eg. Bad CRC, parity, etc.
               ELSE
                   #sb.log.Error_exception_cnt += 1;
               END_IF;

               // Increase communication error counter. if it's a comm.error.
               // then reset the counter.  
               IF #mb_query.stat.error_comm THEN
                   #sb.z.comm_err_cnt += BOOL_TO_USINT(#sb.z.comm_err_cnt < 250);
               ELSE
                   #sb.z.comm_err_cnt := 0;
               END_IF;

               // The error_comm flag is set if x repeating comm.errors occurres.
               #err := #sb.z.comm_err_cnt > #sb.conf.max_comm_error;
               IF #err AND NOT #sb.out.Communication_error THEN
                   // Log the time when the flag is set.
                   #"e" := RD_LOC_T(#sb.log.Disconnected_time);
               END_IF;
               #sb.out.Communication_error := #err;

               // A comm.error will not be displayed before the
               // communication_error flag is set. Other errors will be
               // diplayed once. (NOT comm.error -> normal error)
               #sb.out.Error := #sb.out.Error OR NOT #mb_query.stat.error_comm
               OR #sb.out.Communication_error;

               // err_hold makes the error flag stay true for more then just
               // one plc-scan.
               #sb.z.err_hold := #sb.out.Error;

           ELSIF #mb_query.stat.done THEN // Logging successfully query        
               #sb.log.Done_cnt += 1;
               // One successfully query -> reset fault.
               #sb.out.Communication_error := false;
               #sb.z.comm_err_cnt := 0;
               // Note: #sb.out.error shouldn't be set false at this point.
           END_IF;

           // - If it's this devices has the retry token, (sid_retry = sid_cnt)
           //   a retry has been executed and faild. Then set the retry_finished
           //   flag.
           // - The retry-token will be passed on to the next device with
           //   communication problems when the query loop has reach
           //   the end. (Inside the mb_internal_e)
           // - The library make sure that only one station block with comm.
           //   problems will do retry for each query loop revolution. 
           #mb_query.z.sb.sid_retry_finished :=
           #mb_query.z.sb.sid_retry = #mb_query.z.sb.sid_cnt
           AND #mb_query.stat.error_comm;

           // Only one query in the SB is executed (default). The purpose is
           // to avoid a SB with many queries to occupy the bus for long periodes
           // of time. offset_qid is incread by one when a query has executed
           // given last query didn't resualt in a timeout.
           #sb.z.offset_qid += BOOL_TO_UINT(NOT #mb_query.stat.error_comm);
       END_IF;
   END_REGION

   REGION Middle
       // If all queries for this device has been executed,
       // then reset offset_qid back to the first query.
       IF #sb.z.offset_qid >
           #mb_query.z.run.qid_cnt - #sb.z.header_qid
       THEN
           #sb.z.offset_qid := 1;

           // Also reset error falg, if the last query was successfully.
           IF NOT #sb.z.err_hold THEN
               #sb.out.Error := false;
           END_IF;
           #sb.z.err_hold := false;
       END_IF;

       // If the retry-token point at this device (sid_retry=sid_cnt), and there is
       // no communication problems then pass on the retry-token to the next device.
       // The retry token tell which device with communication problem that should
       // retry establish communication.
       #mb_query.z.sb.sid_retry +=
       BOOL_TO_UINT(#mb_query.z.sb.sid_retry = #mb_query.z.sb.sid_cnt
                    AND NOT #sb.out.Communication_error);
   END_REGION

   REGION Finnish
       // Several condition that resault in passing on the query-token on to the
       // next device. Skipping all or the rest of the queries for this device:              
       #sb.out.Finnish :=
       #mb_query.z.sb.head_recive AND ( // Skip rest of the queries if: ->
       (* *)#sb.z.exec_cnt >= #sb.conf.exec_quantity // Some queries has executed,
       (*           *)// wait for the next loop for the remaining queries.
       (*      *)OR #mb_query.stat.error_comm) // A query resualting in comm.error    
       OR #mb_query.z.sb.head_insert AND ( // Erase a already inserted query if: ->
       (* *)#sb.out.Communication_error // This station has allready comm. problems.
       (*      *)// And, it isn't this devies turn to try again.
       (*      *)AND (#mb_query.z.sb.sid_retry <> #mb_query.z.sb.sid_cnt
       (*           *)// Or, there has allready been a retry attempt on this loop.
       (*           *)OR #mb_query.z.sb.sid_retry_finished) // (reseted in mb_internal_e)     
       (* *)OR #sb.conf.disable    
       (* *)OR #sb.conf.exec_quantity = 0 // Zero => disable station block.
       (* *)OR #sb.conf.read_only // The read_only flag is set, and it's a write query.
       (*      *)AND #mb_query.z.run.write);

       IF #sb.out.Finnish THEN // Reset
           // Go back to the first state in mb_query. New query param. will owerwrite 
           // old once. Note: usual when changing state, there should be condidion 
           // that the state isn't EXEC_QUERY, but head_recive or head_insert is ture,
           // then we know that state isn't EXEC_QUERY.
           #mb_query.z.run.state := #ORIGIN;
           // Set to qid to the next station block.
           #mb_query.z.run.qid := #mb_query.z.run.qid_cnt + 1;
           #sb.z.exec_cnt := 0;

           // If the sb is read only mode and a write query is hit, then skip it
           // and advance to the next query on the next run.
           #sb.z.offset_qid +=
           (* *)BOOL_TO_UINT(#sb.conf.read_only AND #mb_query.z.run.write);        
       END_IF;

       IF #sb.out.Error THEN // The error is forwared to the error output on the ctrl.
           #mb_query.z.sb.error := true;
       END_IF;
   END_REGION
END_FUNCTION

// folder: Library/Modbus/Core/Sequence

FUNCTION_BLOCK "mb_sequence"   // FB21, SCL
{ S7_Optimized_Access := 'TRUE' }
VERSION : 0.1
   VAR_IN_OUT
      sb : "mb_station_block_udt";   // Station block udt
      mb_query : "mb_query";
   END_VAR
   VAR
      Done : Bool;   // All queries has been exec. at least once, and no query has error.
      Error : Bool;   // At least one query has error.
      conf : Struct
         first_state : Int := 32767;   // Init state
      END_STRUCT;
      state : Int := 32767;
      next_state : Int := 32767;   // Will be transfer to state when query finnished
      z : Struct   // Internal variables
         first_scan : Bool := true;
         state_with_error : Int;
         a_query_is_executed : Bool;
      END_STRUCT;
   END_VAR
   VAR_TEMP
      write : Bool;
      exec : Bool;
   END_VAR
BEGIN
   // This FB should be called after a state machine with queries, and
   // be used together with mb_sequence_init, which should be called 
   // at the top of the state machine. The purpose is to make some less
   // important queries be executed less often. Or it can be used to make
   // some queries be executed at a given order.
   // 
   // Features:
   //  - An error on one querie in the state machine will make
   //    #sb.out.error stay true, until the error is solved.
   //  - If #sb.conf.read_only is set, then a state with a write query
   //    will be skipped.
   //  - Handle incrementing the state counter when a query finnish.
   //  - Simple interface for next-query and first-query.
   //  - A Done flag that will be set when all queries in the state 
   //    machine has been executed successfully.

   // Figur out if the current state has a write query.
   CASE #mb_query.mode OF
       5, 6, 15, 16, 201, 202: // Write fc's.
           #write := true;
   END_CASE;

   // A query has executed, and there is a respons from device.
   #exec := #mb_query.Done
   (* *)OR #mb_query.Error AND NOT #mb_query.stat.error_comm;

   IF #sb.out.Communication_error THEN
       IF #conf.first_state <> 32767 THEN
           #state := #conf.first_state;
       END_IF;
       // On a communication error then Done flag will be released.
       #z.a_query_is_executed := #Done := false;

       // Go to next state, if the query in the current state has been
       // executed. (successfully or with error)
       // Or, go to next state if the query in current state is a
       // write query and at the same time the read_only flag is set.
       // (#sb.conf.read_only)
   ELSIF #exec OR #write AND #sb.conf.read_only THEN
       IF #exec THEN
           // Set the error flag, even if it's just one query in
           // the state machine that has an error.
           IF #mb_query.Error AND NOT #mb_query.stat.error_comm THEN
               #Error := true;
               // There may be more than one state with a error, in that
               // case both errors need to be solved before the error flag 
               // is released.
               #z.state_with_error := #state;
           ELSIF #mb_query.Done
               AND #z.state_with_error = #state
           THEN
               // If it's a successful query, and this state is the one
               // that had query with error before, then release the 
               // error flag.
               #Error := false;
           END_IF;
           // All queries has been executed at least once.
           IF #z.a_query_is_executed
               AND #state = #conf.first_state
               AND NOT #Error // No query with error.
           THEN
               #Done := true;
           END_IF;
           #z.a_query_is_executed := true;
       END_IF;
       // Change state
       #state := SEL(G := #next_state = 32767,
                     IN0 := #next_state,
                     IN1 := #state + 1);
   ELSE
       #mb_query.z.sb.seq_release := false;
   END_IF;

   IF #Error THEN
       #sb.z.err_hold := #sb.out.Error := true;
   END_IF;

   #next_state := 32767;
   #z.first_scan := false;
END_FUNCTION_BLOCK

FUNCTION "mb_sequence_init" : Int   // FC7, SCL
{ S7_Optimized_Access := 'TRUE' }
VERSION : 0.1
   VAR_IN_OUT
      sequence : "mb_sequence";
      mb_query : "mb_query";
   END_VAR
BEGIN
   // Block should be called inside CASE OF statement, it will 
   // output the current state.

   // In case there is no query in state that being executed.
   #mb_query.Done := #mb_query.Error := false;

   // Transfer first state in to the current on first scan.
   IF #sequence.z.first_scan 
       AND #sequence.conf.first_state <> 32767
   THEN
       #sequence.state := #sequence.conf.first_state;
   END_IF;

   // The third and fourth digit in state will decide function code
   // while the first and secound is a running number. Eg state 300,
   // 301 and 302 is read holding register states. State 1600 and
   // 1601 are states that write holding registers. And state 400
   // and 401 is reading input register.
   #mb_query.mode := INT_TO_USINT(#sequence.state / 100);

   // Current state.
   #mb_sequence_init := #sequence.state;
END_FUNCTION

// folder: Library/Modbus/Core/Swap

FUNCTION "mb_swap_word" : Int   // FC24, SCL
{ S7_Optimized_Access := 'TRUE' }
VERSION : 0.1
   VAR_INPUT
      start : DInt;   // Start address, 0=Auto
      end : DInt;   // End address, 0=Auto
   END_VAR
   VAR_IN_OUT
      q : "mb_query";
   END_VAR
   VAR_TEMP
      c : Int;
      buffer_lo : DInt;
      buffer_hi : DInt;
      tmp : Word;
   END_VAR
BEGIN
   // Swap bytes in buffer. Every second word is swaped
   // with the one before. from addr #start to addr #end.
   //
   // This function dosen't work for discrete quries !

   IF "mb_internal_s"(start := #start,
                          end := #end,
                          buffer_lo := #buffer_lo,
                          buffer_hi := #buffer_hi,
                          q := #q)
   THEN
       // Swap every secound word with the one before.
       FOR #c := #buffer_lo TO #buffer_hi BY 4 DO
           #tmp.%B0 := #q.z.buffer[#c + 0];
           #tmp.%B1 := #q.z.buffer[#c + 1];
           #q.z.buffer[#c + 0] := #q.z.buffer[#c + 2];
           #q.z.buffer[#c + 1] := #q.z.buffer[#c + 3];
           #q.z.buffer[#c + 2] := #tmp.%B0;
           #q.z.buffer[#c + 3] := #tmp.%B1;
       END_FOR;
       #mb_swap_word := 0;
   ELSE // Error handling.
       #mb_swap_word := WORD_TO_INT(#q.stat.status);
   END_IF;
END_FUNCTION

FUNCTION "mb_little_endian" : Int   // FC28, SCL
{ S7_Optimized_Access := 'TRUE' }
VERSION : 0.1
   VAR_INPUT
      start : DInt;   // Start address, 0=Auto
      end : DInt;   // End address, 0=Auto
   END_VAR
   VAR_IN_OUT
      q : "mb_query";
   END_VAR
   VAR_TEMP
      c : Int;
      buffer_lo : DInt;
      buffer_hi : DInt;
      tmp : Word;
   END_VAR
BEGIN
   // Change bytes four and four in buffer, from big endian
   // to little endian.
   // 
   // This function dosen't work for discrete quries !

   IF "mb_internal_s"(start := #start,
                          end := #end,
                          buffer_lo := #buffer_lo,
                          buffer_hi := #buffer_hi,
                          q := #q)
   THEN
       // Change bytes to little endian.
       FOR #c := #buffer_lo TO #buffer_hi BY 4 DO
           #tmp.%B0 := #q.z.buffer[#c + 0];
           #tmp.%B1 := #q.z.buffer[#c + 1];
           #q.z.buffer[#c + 0] := #q.z.buffer[#c + 3];
           #q.z.buffer[#c + 1] := #q.z.buffer[#c + 2];
           #q.z.buffer[#c + 2] := #tmp.%B1;
           #q.z.buffer[#c + 3] := #tmp.%B0;
       END_FOR;

       #mb_little_endian := 0;
   ELSE // Error handling.
       #mb_little_endian := WORD_TO_INT(#q.stat.status);
   END_IF;
END_FUNCTION

// folder: Library/Modbus/Core/Tcp

FUNCTION_BLOCK "mb_delay"   // FB11, SCL
{ S7_Optimized_Access := 'TRUE' }
VERSION : 0.1
   VAR_INPUT
      delay : Time;
   END_VAR
   VAR_IN_OUT
      mb_query : "mb_query";
   END_VAR
   VAR
      "timer" : TON_TIME;
      halt : Bool;
   END_VAR
BEGIN
   // For use with modbus tcp, so the client dosen't jam a network.
   // The function halt execution of queries for a certain time

   #mb_query.z.run.qid_cnt += 1;  // The timer occupy one qid.

   IF #halt // If the timer has been activated.
       OR #delay = T#0s // #delay = T#0s => Disable function
   THEN
       PRESET_TIMER(PT := #delay, TIMER := #"timer");
       #"timer"(IN := #delay <> T#0s, PT := #delay);
       IF #"timer".Q OR #delay = T#0s THEN
           IF #halt THEN
               #mb_query.conf.halt := #halt := false; // Continue exec.
               RESET_TIMER(#"timer");
           END_IF;
           #mb_query.z.run.qid += BOOL_TO_UINT
           (* *)(#mb_query.z.run.qid = #mb_query.z.run.qid_cnt);
       END_IF;

   ELSIF #mb_query.z.run.qid_cnt = #mb_query.z.run.qid THEN
       #mb_query.conf.halt := #halt := true; // Halt exec.
   END_IF;
END_FUNCTION_BLOCK

FUNCTION_BLOCK "mb_delay_between_queries"   // FB13, SCL
{ S7_Optimized_Access := 'TRUE' }
VERSION : 0.1
   VAR_INPUT
      delay : Time;
   END_VAR
   VAR_IN_OUT
      mb_query : "mb_query";
   END_VAR
   VAR
      "timer" : TON_TIME;
      halt : Bool;
      old_state : UInt;
   END_VAR
   VAR CONSTANT
      ORIGIN : USInt := 0;
   END_VAR
BEGIN
   // For use with modbus tcp, so the client dosen't jam a network.
   // The function halt execution of queries for a certain time
   // not just once, but between every query. There should only be
   // one of this block for each client.

   IF #halt // Is exec. halted?
       OR #delay = T#0s // #delay = T#0s => Disable function.
   THEN
       PRESET_TIMER(PT := #delay, TIMER := #"timer");
       #"timer"(IN := #delay <> T#0s, PT := #delay);
       IF #"timer".Q
           OR #delay = T#0s AND #halt
       THEN
           RESET_TIMER(#"timer");
           #mb_query.conf.halt := #halt := false; // Continue exec.
       END_IF;

   ELSIF #mb_query.z.run.state <> #old_state
       AND #mb_query.z.run.state <> #ORIGIN
   THEN
       // Halt exec. when next query is about to be inserted,
       // but current query will still finish.
       #mb_query.conf.halt := #halt := true; // Halt exec.
   END_IF;
   #old_state := #mb_query.z.run.state;
END_FUNCTION_BLOCK

FUNCTION "mb_tcp_connection_header" : Void   // FC19, SCL
{ S7_Optimized_Access := 'TRUE' }
VERSION : 0.1
   VAR_IN_OUT
      conn : "mb_tcp_connection_udt";   // Connection udt
      ctrl : "mb_tcp_ctrl";   // mb_client_ctrl
      q : "mb_query";   // mb_query
   END_VAR
   VAR CONSTANT
      ORIGIN : USInt := 0;
      INSERT_QUERY : USInt := 1;
      INIT_QUERY : USInt := 2;
      EXEC_QUERY : USInt := 3;
      RECIVE_RESUALT : USInt := 4;
   END_VAR
BEGIN
   // This block need to be placed before the station blocks, for the
   // current tcp-connection.
   //
   // This block together with mb_tcp_connection_foother will manupulate
   // variables in mb_client_ctrl. When a query between header and
   // foother has been inserted, the foother will disconnect and 
   // reconnect to the new ip/port, though only if it's different from
   // the one active.

   // When state is at INIT_QUERY it means that a new query has been
   // inserted. This info is used in tcp-foother, for checking if a query
   // has been inserted between the header and the foother.
   #conn.z.init_at_header := #q.z.run.state = #INIT_QUERY;

   // If set_err is true, all error flags on all sb's will be set to true.
   #q.z.sb.set_err := false; // Default value.

   // Check if current query is bellow.
   #conn.z.qid_bellow := #q.z.run.qid_cnt < #q.z.run.qid;

   IF #q.z.run.state = #RECIVE_RESUALT THEN
       // A new resault has arrived. If correct ip-address and
       // tcp-port. The resualt bellong to this connetion.
       IF #ctrl.ip_addr = #conn.ip
           AND #ctrl.tcp_port = #conn.tcp_port
       THEN
           // Deal with any errors.
           #conn.Error := #q.stat.error;
           IF #q.stat.error THEN
               // Save device/unit with error for easier debugging.
               #conn.Error_unit := UINT_TO_USINT(#q.z.q.mb_addr);
               // Check if it's network (ethernet) problem.
               #q.z.sb.set_err := #conn.Error_network := NOT #ctrl.connected;
           END_IF;
       ELSE
           // If different ip or port, then this resault
           // dosen't bellong to this connection. Block
           // any query from reciving resualt.
           #q.z.run.state := 10;
           // State is set back to RECIVE_RESUALT in the
           // mb_tcp_connection_foother.
       END_IF;
       // Make all quries inside the station blocks be executed right
       // away. This is more efficent then executing one by one query,
       // since it take time to esablish a tcp connection.
       #q.z.sb.exec_all := true;
   END_IF;
END_FUNCTION

FUNCTION "mb_tcp_connection_foother" : Void   // FC21, SCL
{ S7_Optimized_Access := 'TRUE' }
VERSION : 0.1
   VAR_IN_OUT
      conn : "mb_tcp_connection_udt";
      ctrl : "mb_tcp_ctrl";
      q : "mb_query";
   END_VAR
   VAR_TEMP
      equal : Bool;
   END_VAR
   VAR CONSTANT
      ORIGIN : USInt := 0;
      INSERT_QUERY : USInt := 1;
      INIT_QUERY : USInt := 2;
      EXEC_QUERY : USInt := 3;
      RECIVE_RESUALT : USInt := 4;
   END_VAR
BEGIN
   // This fc should be placed after all station blocks
   // for the current tcp-connection-setting.


   // If set_err is true, all error flags on all sb's will be set to true.
   #q.z.sb.set_err := false; // Default value.

   #equal := #conn.tcp_port = #ctrl.tcp_port
   (* *)AND #conn.ip = #ctrl.ip_addr;

   CASE #q.z.run.state OF
       10: // Ten is a blocking-state for reciving resualt, this value is assigned
           // in mb_tcp_connection_header.
           IF #q.z.run.qid_cnt >= #q.z.run.qid
               AND #conn.z.qid_bellow
               AND NOT #equal
           THEN
               // Deadlock handling.
               // It may happen that query bellong to one connection is wating
               // for a resault, but the ip hasen't been changed. Since state
               // is ten, the query will never finnish, and there is a deadlock.
               #q.z.run.state := #ORIGIN; // Back to start, out of deadlock.
               // Set to qid to the next connection.
               #q.z.run.qid := #q.z.run.qid_cnt + 1;
           ELSE
               #q.z.run.state := #RECIVE_RESUALT;
           END_IF;
   END_CASE;

   // ------- Disconnect ------- 
   IF #q.z.run.state = #INIT_QUERY
       AND NOT #conn.z.init_at_header
       AND NOT #equal // IP-address and port.
   THEN
       // If state wasn't INIT_QUERY at header, but it's INIT_QUERY at foother,
       // that means one query has insertet it's parameter inbetween, and it's
       // ready to be executed. If on top of that the ip/port is different from
       // current setting, then we need to disconnect and then reconnect with
       // the new ip/port-settings.

       // Disconnect (reconnect to new ip/port bellow)
       #conn.z.disconnect := #ctrl.conf.disconnect := true;
       // Block mb_client_ctrl from init and exec. the query.
       #q.z.run.state := 11; // (Set back bellow)

       // ------- Resconnect ------- 
   ELSIF #conn.z.disconnect  // This connection-setting, has cmd to disconnect.
       AND #q.stat.status = 16#7000  // Disconnect is finnish.
       // 7000: No job active and no connection established.
   THEN
       // When disconnected, then set new ip and port and reconnect.
       #ctrl.ip_addr := #conn.ip; // New tcp/ip settings.
       #ctrl.tcp_port := #conn.tcp_port;
       // Reconnect.
       #conn.z.disconnect := #ctrl.conf.disconnect := false;
       #q.z.run.state := #INIT_QUERY; // Set back from 11 above.
       GOTO TIMEOUT_OVERRIDE;

   ELSIF #equal THEN
       // ------- No connection (timeout) ------- 
       IF #q.z.run.state <> #EXEC_QUERY
           AND NOT #ctrl.connected
           AND #ctrl.ton_timeout.Q // Timeout connecting.
       THEN
           // Reset, set state back for inserting another query.
           #q.z.run.state := #ORIGIN;
           // Set to qid to the next station block.
           #q.z.run.qid := #q.z.run.qid_cnt + 1;

       ELSE // ------- Set timeout ------- 
           GOTO TIMEOUT_OVERRIDE;
       END_IF;
   END_IF;

   RETURN;

   TIMEOUT_OVERRIDE:
   // Use custom timeout for this connection, if timeout is set.    
   IF #conn.timeout <> T#0s THEN
       #ctrl.override_timeout := #conn.timeout;
   END_IF;
END_FUNCTION

// folder: Library/Modbus/Core/z/z Internal

FUNCTION_BLOCK "mb_internal_b"   // FB6, SCL
{ S7_Optimized_Access := 'FALSE' }
VERSION : 0.1
   VAR
      buffer : Array[0..249] of Byte;
   END_VAR
BEGIN
   (*
   - Buffer for mb_master and modbus_master. (modbus rtu)
   - This block has optimize data access disabled.
   - For rtu, please do not delete this block, even there is no code bellow.
   - This block isn't needed for modbus tcp.
   *)
END_FUNCTION_BLOCK

FUNCTION_BLOCK "mb_internal_e"   // FB7, SCL
{ S7_Optimized_Access := 'TRUE' }
VERSION : 0.1
   VAR_OUTPUT
      Error : Bool;
   END_VAR
   VAR_IN_OUT
      mb_query : "mb_query";
   END_VAR
   VAR
      err_hold : Bool;
   END_VAR
   VAR CONSTANT
      INSERT_QUERY : USInt := 1;
      EXEC_QUERY : USInt := 3;
      RECIVE_RESUALT : USInt := 4;
   END_VAR
BEGIN
   // Internal function - common for both rtu and tcp.

   // Move on to next state when query is finnished.
   IF #mb_query.z.run.state = #EXEC_QUERY 
       AND (#mb_query.stat.error OR #mb_query.stat.done)
   THEN
       #mb_query.z.run.state := #RECIVE_RESUALT;
   END_IF;


   // Anti wind up effect for qid. msg. to devices that they should
   // reset if qid grow bigger then 60000. (See mb_station_block_header)
   #mb_query.z.sb.reset := false;
   IF #mb_query.z.run.qid > 60000 THEN
       #mb_query.z.sb.reset := true;
   END_IF;

   // #error will be keeped true as long there is at least one query that
   // generate a error. 
   IF #mb_query.stat.error
       OR #mb_query.z.sb.error // Pick up error from any sb
   THEN
       #Error := true;
       #err_hold := true;
   END_IF;
   #mb_query.z.sb.error := false;

   // If all queries has been executed,
   IF #mb_query.z.run.qid > #mb_query.z.run.qid_cnt THEN

       // Error handeling (see above)
       IF NOT #err_hold THEN
           #Error := false;
       END_IF;
       #err_hold := false;

       // Start over again on the first query.
       #mb_query.z.run.qid := 1;

       // The retry-id is the device that get to have retry to restoring
       // communication after the error_comm flag is set for the station.
       // When one query loop has occurred the retry id is incremented. 
       #mb_query.z.sb.sid_retry := #mb_query.z.sb.sid_retry + 1;

       // retry_finished is set after one retry has taken place. 
       // The station that has the retry-token only has one try to make 
       // successfully query.
       #mb_query.z.sb.sid_retry_finished := false;
       IF #mb_query.z.sb.sid_retry > #mb_query.z.sb.sid_cnt THEN
           #mb_query.z.sb.sid_retry := 1;
       END_IF;

       // Station id (sid):
       // A sb can do some action, when sid_cnt is equal it's sid.
       // If sid_halt is set true, sid inc. will then stop until it's
       // released. 
       #mb_query.z.sb.sid := #mb_query.z.sb.sid
       (* *)+ BOOL_TO_UINT(NOT #mb_query.z.sb.sid_halt);
       #mb_query.z.sb.sid_halt := false;
       IF #mb_query.z.sb.sid > #mb_query.z.sb.sid_cnt THEN
           #mb_query.z.sb.sid := 1;
       END_IF;
   END_IF;

   #mb_query.z.run.qid_cnt := 0; // (Incremented in mb_query)
   #mb_query.z.sb.sid_cnt := 0; // (Incremented in mb_station_block_header)

   // Default value:
   // 1: Set error flags on all sb's.
   // 2: Makes all (255) queries be executed right away in a sb's.
   #mb_query.z.sb.set_err := #mb_query.z.sb.exec_all := false;
END_FUNCTION_BLOCK

FUNCTION "mb_internal_f" : Void   // FC2, SCL
{ S7_Optimized_Access := 'TRUE' }
VERSION : 0.1
   VAR_IN_OUT
      buffer : "mb_internal_b";
      mb_query : "mb_query";
   END_VAR
   VAR_TEMP
      comm_error : Bool;
   END_VAR
BEGIN
   // Internal function - master footer

   IF #mb_query.stat.error THEN
       // Figur out if it's a communication error.
       // (Handled different from other errors)
       CASE WORD_TO_UINT(#mb_query.stat.status) OF
           16#80C8, // Timeout
           16#80E1, // Parity error
           16#80E2, // Framing error
           16#8380: // Bad CRC 
               #comm_error := true;
       END_CASE;

   ELSIF #mb_query.stat.done // Successful query
       AND NOT #mb_query.z.run.write // A read query.
   THEN
       #mb_query.z.buffer := #buffer.buffer;
   END_IF;

   #mb_query.stat.error_comm :=
   (* *)#mb_query.stat.error AND #comm_error;
END_FUNCTION

FUNCTION "mb_internal_a" : Void   // FC4, SCL
{ S7_Optimized_Access := 'TRUE' }
VERSION : 0.1
   VAR_OUTPUT
      Mode : USInt;
      Data_addr : UDInt;
   END_VAR
   VAR_IN_OUT
      mb_query : "mb_query";
   END_VAR
   VAR_TEMP
      skip : Bool;
   END_VAR
BEGIN
   // Internal function - Modicon convention address.

   #Mode := 0;
   CASE #mb_query.z.q.mode OF
       1, 2, 4, 5, 15:
           IF #mb_query.z.q.data_addr > 9999 THEN
               #Mode := #mb_query.z.q.mode + 100;
               #Data_addr := #mb_query.z.q.data_addr;
               RETURN;
           END_IF;
   END_CASE;
   CASE #mb_query.z.q.mode OF
       1:  // Read output bits
           #Data_addr := 1 + #mb_query.z.q.data_addr;
       2:  // Read input bits
           #Data_addr := 10001 + #mb_query.z.q.data_addr;
       3:  // Read holding reg.
           #Data_addr := 400001 + #mb_query.z.q.data_addr;
       4:  // Read input word
           #Data_addr := 30001 + #mb_query.z.q.data_addr;
       5:  // Writing a single output bit
           #Mode := 1;
           #Data_addr := 1 + #mb_query.z.q.data_addr;
       6:  // Writing a single holding register
           #Mode := 1;
           #Data_addr := 400001 + #mb_query.z.q.data_addr;
       15: // Writing multiple output bits
           #Mode := 2;
           #Data_addr := 1 + #mb_query.z.q.data_addr;
       16: // Writing multiple holding registers
           #Mode := 2;
           #Data_addr := 400001 + #mb_query.z.q.data_addr;
       200..202: // Read and write
           #Mode := #mb_query.z.q.mode - 200;
           #Data_addr := #mb_query.z.q.data_addr;
       ELSE
           #Mode := #mb_query.z.q.mode;
           #Data_addr := #mb_query.z.q.data_addr;
   END_CASE;
END_FUNCTION

FUNCTION "mb_timeout_rtu_calc" : Time   // FC5, SCL
{ S7_Optimized_Access := 'TRUE' }
VERSION : 0.1
   VAR_INPUT
      timeout : Time;
      baud : UDInt;
   END_VAR
   VAR_IN_OUT
      mb_query : "mb_query";
   END_VAR
   VAR_TEMP
      "time" : Time;
      rBytes : Real;
      rBaud : Real;
   END_VAR
BEGIN
   // Automatically adjust timeout for modbus rtu.

   #rBaud := UDINT_TO_REAL(#baud);
   #rBytes := UDINT_TO_REAL(#mb_query.z.run.bytes);
   #"time" :=
   T_CONV
   (REAL_TO_DINT
    (11000 * (19 + #rBytes) / #rBaud * 1.5)) + #timeout;
   #mb_timeout_rtu_calc :=
   LIMIT(MN := T#15ms, 
         IN := #"time",
         MX := T#20s);
   (*
   mb_comm_load require a least 5ms, else a error will be thrown.

   11000 => 11     : Bits: start, data, parity, stop.  
            * 1000 : Seconds to milliseconds
   19    => Fixed bytes in msg: Req: mb_addr, fc, 
            data_addr(2), data_len(2), crc(2), 
            resonse: mb_addr, fc, byte-count, crc(2), 
            start-stop: 6 (about 2 x 28 bits)
   3     => Safty margin
   *)
END_FUNCTION

FUNCTION "mb_internal_s" : Bool   // FC23, SCL
{ S7_Optimized_Access := 'TRUE' }
VERSION : 0.1
   VAR_INPUT
      start : DInt;
      end : DInt;
   END_VAR
   VAR_IN_OUT
      buffer_lo : DInt;
      buffer_hi : DInt;
      q : "mb_query";
   END_VAR
   VAR_TEMP
      tmp : DInt;
   END_VAR
BEGIN
   // Internal function in the library for calculating
   // beginning and end for swapping.
   // 
   // This function dosen't work for discrete quries !

   // Find the beginning in the buffer where swaping should start.
   #buffer_lo := SEL(G := #start = 0,
                     IN0 := (#start - UDINT_TO_DINT(#q.z.q.data_addr)) * 2,
                     IN1 := 0);

